LIN {X -32.888,Y -21.847,Z -39.181,A -90.000,B 90.000,C 0.000} C_DIS
LIN {X -32.646,Y -21.814,Z -39.101,A -90.000,B 90.000,C 0.000} C_DIS
LIN {X -32.451,Y -21.791,Z -39.046,A -90.000,B 90.000,C 0.000} C_DIS
LIN {X -32.080,Y -21.753,Z -38.957,A -90.000,B 90.000,C 0.000} C_DIS
LIN {X -31.853,Y -21.730,Z -38.910,A -90.000,B 90.000,C 0.000} C_DIS
LIN {X -31.718,Y -21.717,Z -38.887,A -90.000,B 90.000,C 0.000} C_DIS
LIN {X -31.508,Y -21.700,Z -38.859,A -90.000,B 90.000,C 0.000} C_DIS
LIN {X -31.116,Y -21.673,Z -38.819,A -90.000,B 90.000,C 0.000} C_DIS
LIN {X -31.063,Y -21.669,Z -38.814,A -90.000,B 90.000,C 0.000} C_DIS
LIN {X -30.892,Y -21.659,Z -38.806,A -90.000,B 90.000,C 0.000} C_DIS
LIN {X -30.823,Y -21.657,Z -38.806,A -90.000,B 90.000,C 0.000} C_DIS
LIN {X -30.549,Y -21.645,Z -38.800,A -90.000,B 90.000,C 0.000} C_DIS
LIN {X -30.055,Y -21.635,Z -38.810,A -90.000,B 90.000,C 0.000} C_DIS
LIN {X -28.776,Y -21.601,Z -38.842,A -90.000,B 90.000,C 0.000} C_DIS
LIN {X -28.195,Y -21.575,Z -38.837,A -90.000,B 90.000,C 0.000} C_DIS
LIN {X -27.943,Y -21.565,Z -38.836,A -90.000,B 90.000,C 0.000} C_DIS
LIN {X -27.045,Y -21.542,Z -38.826,A -90.000,B 90.000,C 0.000} C_DIS
LIN {X -26.882,Y -21.540,Z -38.829,A -90.000,B 90.000,C 0.000} C_DIS
LIN {X -26.670,Y -21.539,Z -38.837,A -90.000,B 90.000,C 0.000} C_DIS
LIN {X -26.459,Y -21.525,Z -38.814,A -90.000,B 90.000,C 0.000} C_DIS
LIN {X -26.307,Y -21.516,Z -38.801,A -90.000,B 90.000,C 0.000} C_DIS
LIN {X -26.029,Y -21.496,Z -38.784,A -90.000,B 90.000,C 0.000} C_DIS
LIN {X -25.788,Y -21.478,Z -38.772,A -90.000,B 90.000,C 0.000} C_DIS
LIN {X -25.199,Y -21.452,Z -38.736,A -90.000,B 90.000,C 0.000} C_DIS
LIN {X -24.907,Y -21.440,Z -38.729,A -90.000,B 90.000,C 0.000} C_DIS
LIN {X -24.488,Y -21.430,Z -38.731,A -90.000,B 90.000,C 0.000} C_DIS
LIN {X -24.339,Y -21.421,Z -38.722,A -90.000,B 90.000,C 0.000} C_DIS
LIN {X -23.648,Y -21.391,Z -38.698,A -90.000,B 90.000,C 0.000} C_DIS
LIN {X -22.784,Y -21.370,Z -38.662,A -90.000,B 90.000,C 0.000} C_DIS
LIN {X -22.360,Y -21.341,Z -38.605,A -90.000,B 90.000,C 0.000} C_DIS
LIN {X -22.032,Y -21.308,Z -38.567,A -90.000,B 90.000,C 0.000} C_DIS
LIN {X -22.032,Y -60.000,Z -38.567,A -90.000,B 90.000,C 0.000} C_DIS
LIN {X -41.599,Y -60.000,Z -38.134,A -90.000,B 90.000,C 0.000} C_DIS
LIN {X -41.599,Y -21.308,Z -38.134,A -90.000,B 90.000,C 0.000} C_DIS
LIN {X -40.454,Y -21.445,Z -38.400,A -90.000,B 90.000,C 0.000} C_DIS
LIN {X -39.852,Y -21.524,Z -38.553,A -90.000,B 90.000,C 0.000} C_DIS
LIN {X -39.336,Y -21.580,Z -38.649,A -90.000,B 90.000,C 0.000} C_DIS
LIN {X -38.632,Y -21.653,Z -38.787,A -90.000,B 90.000,C 0.000} C_DIS
LIN {X -37.790,Y -21.739,Z -38.950,A -90.000,B 90.000,C 0.000} C_DIS
LIN {X -36.979,Y -21.831,Z -39.143,A -90.000,B 90.000,C 0.000} C_DIS
LIN {X -36.858,Y -21.843,Z -39.172,A -90.000,B 90.000,C 0.000} C_DIS
LIN {X -36.574,Y -21.789,Z -38.973,A -90.000,B 90.000,C 0.000} C_DIS
LIN {X -36.491,Y -21.774,Z -38.918,A -90.000,B 90.000,C 0.000} C_DIS
LIN {X -36.292,Y -21.725,Z -38.792,A -90.000,B 90.000,C 0.000} C_DIS
LIN {X -36.111,Y -21.683,Z -38.685,A -90.000,B 90.000,C 0.000} C_DIS
LIN {X -34.878,Y -21.399,Z -38.007,A -90.000,B 90.000,C 0.000} C_DIS
LIN {X -34.510,Y -21.319,Z -37.820,A -90.000,B 90.000,C 0.000} C_DIS
LIN {X -34.454,Y -21.308,Z -37.795,A -90.000,B 90.000,C 0.000} C_DIS
LIN {X -34.454,Y -60.000,Z -37.795,A -90.000,B 90.000,C 0.000} C_DIS
LIN {X -100.614,Y -60.000,Z -38.290,A -90.000,B 90.000,C 0.000} C_DIS
LIN {X -100.614,Y -21.308,Z -38.290,A -90.000,B 90.000,C 0.000} C_DIS
LIN {X -100.205,Y -21.414,Z -38.194,A -90.000,B 90.000,C 0.000} C_DIS
LIN {X -100.106,Y -21.441,Z -38.173,A -90.000,B 90.000,C 0.000} C_DIS
LIN {X -100.009,Y -21.463,Z -38.155,A -90.000,B 90.000,C 0.000} C_DIS
LIN {X -99.788,Y -21.508,Z -38.090,A -90.000,B 90.000,C 0.000} C_DIS
LIN {X -99.614,Y -21.546,Z -38.045,A -90.000,B 90.000,C 0.000} C_DIS
LIN {X -99.380,Y -21.597,Z -37.989,A -90.000,B 90.000,C 0.000} C_DIS
LIN {X -99.127,Y -21.649,Z -37.935,A -90.000,B 90.000,C 0.000} C_DIS
LIN {X -98.699,Y -21.744,Z -37.869,A -90.000,B 90.000,C 0.000} C_DIS
LIN {X -98.267,Y -21.842,Z -37.814,A -90.000,B 90.000,C 0.000} C_DIS
LIN {X -98.126,Y -21.876,Z -37.800,A -90.000,B 90.000,C 0.000} C_DIS
LIN {X -98.086,Y -21.872,Z -37.753,A -90.000,B 90.000,C 0.000} C_DIS
LIN {X -98.019,Y -21.862,Z -37.682,A -90.000,B 90.000,C 0.000} C_DIS
LIN {X -97.690,Y -21.825,Z -37.351,A -90.000,B 90.000,C 0.000} C_DIS
LIN {X -97.548,Y -21.812,Z -37.215,A -90.000,B 90.000,C 0.000} C_DIS
LIN {X -97.502,Y -21.804,Z -37.162,A -90.000,B 90.000,C 0.000} C_DIS
LIN {X -97.462,Y -21.795,Z -37.117,A -90.000,B 90.000,C 0.000} C_DIS
LIN {X -97.361,Y -21.778,Z -37.014,A -90.000,B 90.000,C 0.000} C_DIS
LIN {X -97.077,Y -21.736,Z -36.733,A -90.000,B 90.000,C 0.000} C_DIS
LIN {X -96.910,Y -21.718,Z -36.582,A -90.000,B 90.000,C 0.000} C_DIS
LIN {X -96.744,Y -21.701,Z -36.444,A -90.000,B 90.000,C 0.000} C_DIS
LIN {X -96.611,Y -21.685,Z -36.336,A -90.000,B 90.000,C 0.000} C_DIS
LIN {X -96.274,Y -21.633,Z -36.025,A -90.000,B 90.000,C 0.000} C_DIS
LIN {X -96.149,Y -21.616,Z -35.917,A -90.000,B 90.000,C 0.000} C_DIS
LIN {X -96.043,Y -21.602,Z -35.833,A -90.000,B 90.000,C 0.000} C_DIS
LIN {X -95.731,Y -21.565,Z -35.597,A -90.000,B 90.000,C 0.000} C_DIS
LIN {X -95.458,Y -21.538,Z -35.389,A -90.000,B 90.000,C 0.000} C_DIS
LIN {X -95.333,Y -21.527,Z -35.300,A -90.000,B 90.000,C 0.000} C_DIS
LIN {X -95.028,Y -21.504,Z -35.104,A -90.000,B 90.000,C 0.000} C_DIS
LIN {X -94.893,Y -21.487,Z -35.002,A -90.000,B 90.000,C 0.000} C_DIS
LIN {X -94.794,Y -21.476,Z -34.928,A -90.000,B 90.000,C 0.000} C_DIS
LIN {X -94.672,Y -21.461,Z -34.843,A -90.000,B 90.000,C 0.000} C_DIS
LIN {X -94.553,Y -21.452,Z -34.767,A -90.000,B 90.000,C 0.000} C_DIS
LIN {X -94.476,Y -21.447,Z -34.719,A -90.000,B 90.000,C 0.000} C_DIS
LIN {X -94.315,Y -21.438,Z -34.624,A -90.000,B 90.000,C 0.000} C_DIS
LIN {X -94.176,Y -21.543,Z -34.477,A -90.000,B 90.000,C 0.000} C_DIS
LIN {X -94.101,Y -21.597,Z -34.407,A -90.000,B 90.000,C 0.000} C_DIS
LIN {X -94.045,Y -21.640,Z -34.344,A -90.000,B 90.000,C 0.000} C_DIS
LIN {X -93.974,Y -21.686,Z -34.273,A -90.000,B 90.000,C 0.000} C_DIS
LIN {X -93.825,Y -21.782,Z -34.136,A -90.000,B 90.000,C 0.000} C_DIS
LIN {X -93.634,Y -21.882,Z -33.989,A -90.000,B 90.000,C 0.000} C_DIS
LIN {X -93.528,Y -21.938,Z -33.912,A -90.000,B 90.000,C 0.000} C_DIS
LIN {X -93.397,Y -21.998,Z -33.825,A -90.000,B 90.000,C 0.000} C_DIS
LIN {X -93.347,Y -22.020,Z -33.794,A -90.000,B 90.000,C 0.000} C_DIS
LIN {X -93.262,Y -22.063,Z -33.743,A -90.000,B 90.000,C 0.000} C_DIS
LIN {X -93.192,Y -22.098,Z -33.703,A -90.000,B 90.000,C 0.000} C_DIS
LIN {X -93.048,Y -22.171,Z -33.612,A -90.000,B 90.000,C 0.000} C_DIS
LIN {X -92.988,Y -22.202,Z -33.559,A -90.000,B 90.000,C 0.000} C_DIS
LIN {X -92.889,Y -22.249,Z -33.478,A -90.000,B 90.000,C 0.000} C_DIS
LIN {X -92.767,Y -22.303,Z -33.387,A -90.000,B 90.000,C 0.000} C_DIS
LIN {X -92.764,Y -22.310,Z -33.201,A -90.000,B 90.000,C 0.000} C_DIS
LIN {X -92.753,Y -22.312,Z -33.050,A -90.000,B 90.000,C 0.000} C_DIS
LIN {X -92.734,Y -22.314,Z -32.891,A -90.000,B 90.000,C 0.000} C_DIS
LIN {X -92.716,Y -22.316,Z -32.752,A -90.000,B 90.000,C 0.000} C_DIS
LIN {X -92.695,Y -22.319,Z -32.637,A -90.000,B 90.000,C 0.000} C_DIS
LIN {X -92.629,Y -22.333,Z -32.322,A -90.000,B 90.000,C 0.000} C_DIS
LIN {X -92.598,Y -22.336,Z -32.198,A -90.000,B 90.000,C 0.000} C_DIS
LIN {X -92.561,Y -22.339,Z -32.070,A -90.000,B 90.000,C 0.000} C_DIS
LIN {X -92.530,Y -22.340,Z -31.975,A -90.000,B 90.000,C 0.000} C_DIS
LIN {X -92.451,Y -22.340,Z -31.766,A -90.000,B 90.000,C 0.000} C_DIS
LIN {X -92.397,Y -22.342,Z -31.640,A -90.000,B 90.000,C 0.000} C_DIS
LIN {X -92.293,Y -22.347,Z -31.422,A -90.000,B 90.000,C 0.000} C_DIS
LIN {X -92.165,Y -22.356,Z -31.181,A -90.000,B 90.000,C 0.000} C_DIS
LIN {X -92.072,Y -22.354,Z -31.025,A -90.000,B 90.000,C 0.000} C_DIS
LIN {X -92.020,Y -22.354,Z -30.944,A -90.000,B 90.000,C 0.000} C_DIS
LIN {X -91.933,Y -22.351,Z -30.824,A -90.000,B 90.000,C 0.000} C_DIS
LIN {X -91.750,Y -22.350,Z -30.588,A -90.000,B 90.000,C 0.000} C_DIS
LIN {X -91.667,Y -22.356,Z -30.485,A -90.000,B 90.000,C 0.000} C_DIS
LIN {X -91.552,Y -22.367,Z -30.354,A -90.000,B 90.000,C 0.000} C_DIS
LIN {X -91.426,Y -22.379,Z -30.212,A -90.000,B 90.000,C 0.000} C_DIS
LIN {X -91.373,Y -22.380,Z -30.154,A -90.000,B 90.000,C 0.000} C_DIS
LIN {X -91.227,Y -22.374,Z -29.968,A -90.000,B 90.000,C 0.000} C_DIS
LIN {X -91.132,Y -22.363,Z -29.854,A -90.000,B 90.000,C 0.000} C_DIS
LIN {X -91.028,Y -22.353,Z -29.740,A -90.000,B 90.000,C 0.000} C_DIS
LIN {X -90.920,Y -22.337,Z -29.632,A -90.000,B 90.000,C 0.000} C_DIS
LIN {X -90.736,Y -22.311,Z -29.456,A -90.000,B 90.000,C 0.000} C_DIS
LIN {X -90.615,Y -22.290,Z -29.351,A -90.000,B 90.000,C 0.000} C_DIS
LIN {X -90.528,Y -22.277,Z -29.280,A -90.000,B 90.000,C 0.000} C_DIS
LIN {X -90.420,Y -22.270,Z -29.195,A -90.000,B 90.000,C 0.000} C_DIS
LIN {X -90.287,Y -22.263,Z -29.095,A -90.000,B 90.000,C 0.000} C_DIS
LIN {X -90.131,Y -22.249,Z -28.995,A -90.000,B 90.000,C 0.000} C_DIS
LIN {X -90.003,Y -22.240,Z -28.917,A -90.000,B 90.000,C 0.000} C_DIS
LIN {X -89.988,Y -22.176,Z -28.780,A -90.000,B 90.000,C 0.000} C_DIS
LIN {X -89.968,Y -22.121,Z -28.658,A -90.000,B 90.000,C 0.000} C_DIS
LIN {X -89.961,Y -22.105,Z -28.627,A -90.000,B 90.000,C 0.000} C_DIS
LIN {X -89.926,Y -22.035,Z -28.465,A -90.000,B 90.000,C 0.000} C_DIS
LIN {X -89.879,Y -21.950,Z -28.270,A -90.000,B 90.000,C 0.000} C_DIS
LIN {X -89.848,Y -21.896,Z -28.172,A -90.000,B 90.000,C 0.000} C_DIS
LIN {X -89.820,Y -21.853,Z -28.089,A -90.000,B 90.000,C 0.000} C_DIS
LIN {X -89.771,Y -21.787,Z -27.950,A -90.000,B 90.000,C 0.000} C_DIS
LIN {X -89.722,Y -21.730,Z -27.825,A -90.000,B 90.000,C 0.000} C_DIS
LIN {X -89.648,Y -21.664,Z -27.633,A -90.000,B 90.000,C 0.000} C_DIS
LIN {X -89.586,Y -21.616,Z -27.488,A -90.000,B 90.000,C 0.000} C_DIS
LIN {X -89.533,Y -21.577,Z -27.378,A -90.000,B 90.000,C 0.000} C_DIS
LIN {X -89.338,Y -21.426,Z -27.003,A -90.000,B 90.000,C 0.000} C_DIS
LIN {X -89.314,Y -21.412,Z -26.959,A -90.000,B 90.000,C 0.000} C_DIS
LIN {X -89.215,Y -21.354,Z -26.785,A -90.000,B 90.000,C 0.000} C_DIS
LIN {X -89.141,Y -21.308,Z -26.675,A -90.000,B 90.000,C 0.000} C_DIS
LIN {X -89.043,Y -21.258,Z -26.529,A -90.000,B 90.000,C 0.000} C_DIS
LIN {X -88.953,Y -21.197,Z -26.391,A -90.000,B 90.000,C 0.000} C_DIS
LIN {X -88.870,Y -21.132,Z -26.262,A -90.000,B 90.000,C 0.000} C_DIS
LIN {X -88.725,Y -21.011,Z -26.027,A -90.000,B 90.000,C 0.000} C_DIS
LIN {X -88.663,Y -20.954,Z -25.922,A -90.000,B 90.000,C 0.000} C_DIS
LIN {X -88.608,Y -20.898,Z -25.824,A -90.000,B 90.000,C 0.000} C_DIS
LIN {X -88.559,Y -20.843,Z -25.734,A -90.000,B 90.000,C 0.000} C_DIS
LIN {X -88.517,Y -20.789,Z -25.652,A -90.000,B 90.000,C 0.000} C_DIS
LIN {X -88.482,Y -20.735,Z -25.576,A -90.000,B 90.000,C 0.000} C_DIS
LIN {X -88.452,Y -20.682,Z -25.509,A -90.000,B 90.000,C 0.000} C_DIS
LIN {X -88.429,Y -20.631,Z -25.448,A -90.000,B 90.000,C 0.000} C_DIS
LIN {X -88.405,Y -20.555,Z -25.369,A -90.000,B 90.000,C 0.000} C_DIS
LIN {X -88.394,Y -20.481,Z -25.306,A -90.000,B 90.000,C 0.000} C_DIS
LIN {X -88.394,Y -20.432,Z -25.273,A -90.000,B 90.000,C 0.000} C_DIS
LIN {X -88.405,Y -20.361,Z -25.234,A -90.000,B 90.000,C 0.000} C_DIS
LIN {X -88.411,Y -20.338,Z -25.225,A -90.000,B 90.000,C 0.000} C_DIS
LIN {X -88.427,Y -20.293,Z -25.210,A -90.000,B 90.000,C 0.000} C_DIS
LIN {X -88.461,Y -20.226,Z -25.199,A -90.000,B 90.000,C 0.000} C_DIS
LIN {X -88.490,Y -20.182,Z -25.200,A -90.000,B 90.000,C 0.000} C_DIS
LIN {X -88.542,Y -20.119,Z -25.211,A -90.000,B 90.000,C 0.000} C_DIS
LIN {X -88.583,Y -20.078,Z -25.225,A -90.000,B 90.000,C 0.000} C_DIS
LIN {X -88.628,Y -20.037,Z -25.245,A -90.000,B 90.000,C 0.000} C_DIS
LIN {X -88.678,Y -20.006,Z -25.270,A -90.000,B 90.000,C 0.000} C_DIS
LIN {X -88.732,Y -20.009,Z -25.301,A -90.000,B 90.000,C 0.000} C_DIS
LIN {X -88.853,Y -20.031,Z -25.377,A -90.000,B 90.000,C 0.000} C_DIS
LIN {X -88.919,Y -20.049,Z -25.422,A -90.000,B 90.000,C 0.000} C_DIS
LIN {X -89.063,Y -20.093,Z -25.526,A -90.000,B 90.000,C 0.000} C_DIS
LIN {X -89.222,Y -20.146,Z -25.648,A -90.000,B 90.000,C 0.000} C_DIS
LIN {X -89.306,Y -20.178,Z -25.715,A -90.000,B 90.000,C 0.000} C_DIS
LIN {X -89.577,Y -20.289,Z -25.941,A -90.000,B 90.000,C 0.000} C_DIS
LIN {X -89.773,Y -20.364,Z -26.110,A -90.000,B 90.000,C 0.000} C_DIS
LIN {X -89.979,Y -20.452,Z -26.292,A -90.000,B 90.000,C 0.000} C_DIS
LIN {X -90.194,Y -20.540,Z -26.487,A -90.000,B 90.000,C 0.000} C_DIS
LIN {X -90.418,Y -20.616,Z -26.694,A -90.000,B 90.000,C 0.000} C_DIS
LIN {X -90.649,Y -20.710,Z -26.911,A -90.000,B 90.000,C 0.000} C_DIS
LIN {X -90.887,Y -20.817,Z -27.138,A -90.000,B 90.000,C 0.000} C_DIS
LIN {X -91.130,Y -20.936,Z -27.373,A -90.000,B 90.000,C 0.000} C_DIS
LIN {X -91.378,Y -21.051,Z -27.616,A -90.000,B 90.000,C 0.000} C_DIS
LIN {X -91.630,Y -21.155,Z -27.865,A -90.000,B 90.000,C 0.000} C_DIS
LIN {X -91.884,Y -21.238,Z -28.119,A -90.000,B 90.000,C 0.000} C_DIS
LIN {X -92.140,Y -21.317,Z -28.378,A -90.000,B 90.000,C 0.000} C_DIS
LIN {X -92.396,Y -21.378,Z -28.640,A -90.000,B 90.000,C 0.000} C_DIS
LIN {X -92.653,Y -21.409,Z -28.905,A -90.000,B 90.000,C 0.000} C_DIS
LIN {X -92.908,Y -21.422,Z -29.171,A -90.000,B 90.000,C 0.000} C_DIS
LIN {X -93.160,Y -21.434,Z -29.437,A -90.000,B 90.000,C 0.000} C_DIS
LIN {X -93.410,Y -21.433,Z -29.703,A -90.000,B 90.000,C 0.000} C_DIS
LIN {X -93.655,Y -21.410,Z -29.966,A -90.000,B 90.000,C 0.000} C_DIS
LIN {X -93.895,Y -21.378,Z -30.227,A -90.000,B 90.000,C 0.000} C_DIS
LIN {X -94.129,Y -21.339,Z -30.485,A -90.000,B 90.000,C 0.000} C_DIS
LIN {X -94.356,Y -21.286,Z -30.737,A -90.000,B 90.000,C 0.000} C_DIS
LIN {X -94.575,Y -21.223,Z -30.984,A -90.000,B 90.000,C 0.000} C_DIS
LIN {X -94.785,Y -21.178,Z -31.223,A -90.000,B 90.000,C 0.000} C_DIS
LIN {X -94.984,Y -21.118,Z -31.455,A -90.000,B 90.000,C 0.000} C_DIS
LIN {X -95.173,Y -21.054,Z -31.678,A -90.000,B 90.000,C 0.000} C_DIS
LIN {X -95.350,Y -21.002,Z -31.891,A -90.000,B 90.000,C 0.000} C_DIS
LIN {X -95.514,Y -20.945,Z -32.093,A -90.000,B 90.000,C 0.000} C_DIS
LIN {X -95.664,Y -20.878,Z -32.284,A -90.000,B 90.000,C 0.000} C_DIS
LIN {X -95.733,Y -20.843,Z -32.374,A -90.000,B 90.000,C 0.000} C_DIS
LIN {X -95.860,Y -20.778,Z -32.544,A -90.000,B 90.000,C 0.000} C_DIS
LIN {X -95.971,Y -20.725,Z -32.700,A -90.000,B 90.000,C 0.000} C_DIS
LIN {X -96.064,Y -20.677,Z -32.840,A -90.000,B 90.000,C 0.000} C_DIS
LIN {X -96.139,Y -20.634,Z -32.964,A -90.000,B 90.000,C 0.000} C_DIS
LIN {X -96.195,Y -20.598,Z -33.070,A -90.000,B 90.000,C 0.000} C_DIS
LIN {X -96.215,Y -20.583,Z -33.116,A -90.000,B 90.000,C 0.000} C_DIS
LIN {X -96.240,Y -20.564,Z -33.194,A -90.000,B 90.000,C 0.000} C_DIS
LIN {X -96.245,Y -20.558,Z -33.239,A -90.000,B 90.000,C 0.000} C_DIS
LIN {X -96.241,Y -20.558,Z -33.263,A -90.000,B 90.000,C 0.000} C_DIS
LIN {X -96.237,Y -20.560,Z -33.273,A -90.000,B 90.000,C 0.000} C_DIS
LIN {X -96.224,Y -20.567,Z -33.288,A -90.000,B 90.000,C 0.000} C_DIS
LIN {X -96.216,Y -20.572,Z -33.294,A -90.000,B 90.000,C 0.000} C_DIS
LIN {X -96.181,Y -20.594,Z -33.303,A -90.000,B 90.000,C 0.000} C_DIS
LIN {X -96.150,Y -20.614,Z -33.301,A -90.000,B 90.000,C 0.000} C_DIS
LIN {X -96.113,Y -20.638,Z -33.294,A -90.000,B 90.000,C 0.000} C_DIS
LIN {X -96.070,Y -20.666,Z -33.280,A -90.000,B 90.000,C 0.000} C_DIS
LIN {X -95.963,Y -20.736,Z -33.235,A -90.000,B 90.000,C 0.000} C_DIS
LIN {X -95.830,Y -20.820,Z -33.163,A -90.000,B 90.000,C 0.000} C_DIS
LIN {X -95.668,Y -20.912,Z -33.065,A -90.000,B 90.000,C 0.000} C_DIS
LIN {X -95.477,Y -21.008,Z -32.939,A -90.000,B 90.000,C 0.000} C_DIS
LIN {X -95.257,Y -21.115,Z -32.784,A -90.000,B 90.000,C 0.000} C_DIS
LIN {X -95.005,Y -21.249,Z -32.600,A -90.000,B 90.000,C 0.000} C_DIS
LIN {X -94.867,Y -21.308,Z -32.496,A -90.000,B 90.000,C 0.000} C_DIS
LIN {X -94.735,Y -21.374,Z -32.395,A -90.000,B 90.000,C 0.000} C_DIS
LIN {X -94.474,Y -21.482,Z -32.210,A -90.000,B 90.000,C 0.000} C_DIS
LIN {X -94.461,Y -21.488,Z -32.201,A -90.000,B 90.000,C 0.000} C_DIS
LIN {X -94.382,Y -21.488,Z -31.861,A -90.000,B 90.000,C 0.000} C_DIS
LIN {X -94.318,Y -21.493,Z -31.618,A -90.000,B 90.000,C 0.000} C_DIS
LIN {X -94.247,Y -21.487,Z -31.407,A -90.000,B 90.000,C 0.000} C_DIS
LIN {X -94.177,Y -21.484,Z -31.221,A -90.000,B 90.000,C 0.000} C_DIS
LIN {X -94.106,Y -21.482,Z -31.041,A -90.000,B 90.000,C 0.000} C_DIS
LIN {X -94.015,Y -21.484,Z -30.835,A -90.000,B 90.000,C 0.000} C_DIS
LIN {X -93.966,Y -21.486,Z -30.734,A -90.000,B 90.000,C 0.000} C_DIS
LIN {X -93.872,Y -21.482,Z -30.551,A -90.000,B 90.000,C 0.000} C_DIS
LIN {X -93.807,Y -21.480,Z -30.436,A -90.000,B 90.000,C 0.000} C_DIS
LIN {X -93.713,Y -21.472,Z -30.276,A -90.000,B 90.000,C 0.000} C_DIS
LIN {X -93.592,Y -21.465,Z -30.076,A -90.000,B 90.000,C 0.000} C_DIS
LIN {X -93.524,Y -21.465,Z -29.969,A -90.000,B 90.000,C 0.000} C_DIS
LIN {X -93.480,Y -21.467,Z -29.903,A -90.000,B 90.000,C 0.000} C_DIS
LIN {X -93.350,Y -21.464,Z -29.726,A -90.000,B 90.000,C 0.000} C_DIS
LIN {X -93.271,Y -21.464,Z -29.624,A -90.000,B 90.000,C 0.000} C_DIS
LIN {X -93.117,Y -21.449,Z -29.439,A -90.000,B 90.000,C 0.000} C_DIS
LIN {X -93.016,Y -21.442,Z -29.324,A -90.000,B 90.000,C 0.000} C_DIS
LIN {X -92.865,Y -21.435,Z -29.167,A -90.000,B 90.000,C 0.000} C_DIS
LIN {X -92.717,Y -21.430,Z -29.015,A -90.000,B 90.000,C 0.000} C_DIS
LIN {X -92.650,Y -21.420,Z -28.936,A -90.000,B 90.000,C 0.000} C_DIS
LIN {X -92.474,Y -21.391,Z -28.734,A -90.000,B 90.000,C 0.000} C_DIS
LIN {X -92.283,Y -21.358,Z -28.541,A -90.000,B 90.000,C 0.000} C_DIS
LIN {X -92.197,Y -21.344,Z -28.455,A -90.000,B 90.000,C 0.000} C_DIS
LIN {X -92.033,Y -21.308,Z -28.310,A -90.000,B 90.000,C 0.000} C_DIS
LIN {X -92.033,Y -60.000,Z -28.310,A -90.000,B 90.000,C 0.000} C_DIS
LIN {X -106.753,Y -60.000,Z -42.835,A -90.000,B 90.000,C 0.000} C_DIS
LIN {X -106.753,Y -21.308,Z -42.835,A -90.000,B 90.000,C 0.000} C_DIS
LIN {X -106.698,Y -21.320,Z -42.690,A -90.000,B 90.000,C 0.000} C_DIS
LIN {X -106.625,Y -21.329,Z -42.511,A -90.000,B 90.000,C 0.000} C_DIS
LIN {X -106.563,Y -21.338,Z -42.376,A -90.000,B 90.000,C 0.000} C_DIS
LIN {X -106.515,Y -21.344,Z -42.278,A -90.000,B 90.000,C 0.000} C_DIS
LIN {X -106.418,Y -21.361,Z -42.101,A -90.000,B 90.000,C 0.000} C_DIS
LIN {X -106.303,Y -21.371,Z -41.904,A -90.000,B 90.000,C 0.000} C_DIS
LIN {X -106.128,Y -21.381,Z -41.620,A -90.000,B 90.000,C 0.000} C_DIS
LIN {X -106.072,Y -21.384,Z -41.530,A -90.000,B 90.000,C 0.000} C_DIS
LIN {X -105.932,Y -21.384,Z -41.327,A -90.000,B 90.000,C 0.000} C_DIS
LIN {X -105.884,Y -21.388,Z -41.261,A -90.000,B 90.000,C 0.000} C_DIS
LIN {X -105.762,Y -21.391,Z -41.111,A -90.000,B 90.000,C 0.000} C_DIS
LIN {X -105.660,Y -21.396,Z -40.990,A -90.000,B 90.000,C 0.000} C_DIS
LIN {X -105.461,Y -21.388,Z -40.772,A -90.000,B 90.000,C 0.000} C_DIS
LIN {X -105.340,Y -21.384,Z -40.641,A -90.000,B 90.000,C 0.000} C_DIS
LIN {X -105.188,Y -21.379,Z -40.480,A -90.000,B 90.000,C 0.000} C_DIS
LIN {X -105.077,Y -21.369,Z -40.379,A -90.000,B 90.000,C 0.000} C_DIS
LIN {X -104.931,Y -21.359,Z -40.252,A -90.000,B 90.000,C 0.000} C_DIS
LIN {X -104.638,Y -21.339,Z -40.023,A -90.000,B 90.000,C 0.000} C_DIS
LIN {X -104.496,Y -21.324,Z -39.921,A -90.000,B 90.000,C 0.000} C_DIS
LIN {X -104.322,Y -21.308,Z -39.805,A -90.000,B 90.000,C 0.000} C_DIS
LIN {X -104.322,Y -60.000,Z -39.805,A -90.000,B 90.000,C 0.000} C_DIS
LIN {X -105.044,Y -60.000,Z -54.822,A -90.000,B 90.000,C 0.000} C_DIS
LIN {X -105.044,Y -21.308,Z -54.822,A -90.000,B 90.000,C 0.000} C_DIS
LIN {X -105.069,Y -21.321,Z -54.621,A -90.000,B 90.000,C 0.000} C_DIS
LIN {X -105.095,Y -21.338,Z -54.365,A -90.000,B 90.000,C 0.000} C_DIS
LIN {X -105.108,Y -21.349,Z -54.203,A -90.000,B 90.000,C 0.000} C_DIS
LIN {X -105.120,Y -21.370,Z -53.971,A -90.000,B 90.000,C 0.000} C_DIS
LIN {X -105.123,Y -21.397,Z -53.738,A -90.000,B 90.000,C 0.000} C_DIS
LIN {X -105.123,Y -21.401,Z -53.704,A -90.000,B 90.000,C 0.000} C_DIS
LIN {X -105.093,Y -21.442,Z -53.157,A -90.000,B 90.000,C 0.000} C_DIS
LIN {X -105.069,Y -21.467,Z -52.818,A -90.000,B 90.000,C 0.000} C_DIS
LIN {X -105.063,Y -21.473,Z -52.761,A -90.000,B 90.000,C 0.000} C_DIS
LIN {X -105.048,Y -21.477,Z -52.667,A -90.000,B 90.000,C 0.000} C_DIS
LIN {X -105.149,Y -21.407,Z -52.427,A -90.000,B 90.000,C 0.000} C_DIS
LIN {X -105.259,Y -21.331,Z -52.151,A -90.000,B 90.000,C 0.000} C_DIS
LIN {X -105.294,Y -21.308,Z -52.064,A -90.000,B 90.000,C 0.000} C_DIS
LIN {X -105.294,Y -60.000,Z -52.064,A -90.000,B 90.000,C 0.000} C_DIS
LIN {X -106.298,Y -60.000,Z -243.561,A -90.000,B 90.000,C 0.000} C_DIS
LIN {X -106.298,Y -21.308,Z -243.561,A -90.000,B 90.000,C 0.000} C_DIS
LIN {X -103.088,Y -21.308,Z -241.440,A -90.000,B 90.000,C 0.000} C_DIS
LIN {X -99.816,Y -21.308,Z -239.308,A -90.000,B 90.000,C 0.000} C_DIS
LIN {X -95.252,Y -21.308,Z -236.320,A -90.000,B 90.000,C 0.000} C_DIS
LIN {X -91.143,Y -21.308,Z -233.668,A -90.000,B 90.000,C 0.000} C_DIS
LIN {X -87.088,Y -21.308,Z -231.059,A -90.000,B 90.000,C 0.000} C_DIS
LIN {X -82.371,Y -21.308,Z -228.080,A -90.000,B 90.000,C 0.000} C_DIS
LIN {X -81.805,Y -21.308,Z -227.726,A -90.000,B 90.000,C 0.000} C_DIS
LIN {X -78.607,Y -21.308,Z -225.688,A -90.000,B 90.000,C 0.000} C_DIS
LIN {X -73.743,Y -21.308,Z -222.667,A -90.000,B 90.000,C 0.000} C_DIS
LIN {X -72.906,Y -21.308,Z -222.152,A -90.000,B 90.000,C 0.000} C_DIS
LIN {X -70.393,Y -21.308,Z -220.553,A -90.000,B 90.000,C 0.000} C_DIS
LIN {X -65.618,Y -21.308,Z -217.528,A -90.000,B 90.000,C 0.000} C_DIS
LIN {X -62.348,Y -21.308,Z -215.481,A -90.000,B 90.000,C 0.000} C_DIS
LIN {X -57.206,Y -21.308,Z -212.204,A -90.000,B 90.000,C 0.000} C_DIS
LIN {X -54.876,Y -21.308,Z -210.688,A -90.000,B 90.000,C 0.000} C_DIS
LIN {X -53.612,Y -21.308,Z -209.828,A -90.000,B 90.000,C 0.000} C_DIS
LIN {X -51.750,Y -21.308,Z -208.571,A -90.000,B 90.000,C 0.000} C_DIS
LIN {X -48.408,Y -21.308,Z -206.325,A -90.000,B 90.000,C 0.000} C_DIS
LIN {X -43.930,Y -21.308,Z -203.053,A -90.000,B 90.000,C 0.000} C_DIS
LIN {X -43.271,Y -21.308,Z -202.576,A -90.000,B 90.000,C 0.000} C_DIS
LIN {X -41.226,Y -21.308,Z -200.972,A -90.000,B 90.000,C 0.000} C_DIS
LIN {X -38.879,Y -21.308,Z -199.146,A -90.000,B 90.000,C 0.000} C_DIS
LIN {X -36.934,Y -21.308,Z -197.549,A -90.000,B 90.000,C 0.000} C_DIS
LIN {X -35.130,Y -21.308,Z -196.075,A -90.000,B 90.000,C 0.000} C_DIS
LIN {X -34.778,Y -21.308,Z -195.785,A -90.000,B 90.000,C 0.000} C_DIS
LIN {X -31.882,Y -21.308,Z -193.355,A -90.000,B 90.000,C 0.000} C_DIS
LIN {X -29.706,Y -21.308,Z -191.547,A -90.000,B 90.000,C 0.000} C_DIS
LIN {X -28.831,Y -21.308,Z -190.838,A -90.000,B 90.000,C 0.000} C_DIS
LIN {X -26.880,Y -21.308,Z -189.191,A -90.000,B 90.000,C 0.000} C_DIS
LIN {X -25.951,Y -21.308,Z -188.426,A -90.000,B 90.000,C 0.000} C_DIS
LIN {X -24.127,Y -21.308,Z -186.810,A -90.000,B 90.000,C 0.000} C_DIS
LIN {X -23.356,Y -21.308,Z -186.146,A -90.000,B 90.000,C 0.000} C_DIS
LIN {X -21.765,Y -21.308,Z -184.625,A -90.000,B 90.000,C 0.000} C_DIS
LIN {X -20.866,Y -21.308,Z -183.794,A -90.000,B 90.000,C 0.000} C_DIS
LIN {X -19.977,Y -21.308,Z -182.891,A -90.000,B 90.000,C 0.000} C_DIS
LIN {X -18.317,Y -21.308,Z -181.146,A -90.000,B 90.000,C 0.000} C_DIS
LIN {X -17.573,Y -21.308,Z -180.310,A -90.000,B 90.000,C 0.000} C_DIS
LIN {X -16.056,Y -21.308,Z -178.540,A -90.000,B 90.000,C 0.000} C_DIS
LIN {X -15.581,Y -21.308,Z -177.947,A -90.000,B 90.000,C 0.000} C_DIS
LIN {X -13.815,Y -21.308,Z -175.626,A -90.000,B 90.000,C 0.000} C_DIS
LIN {X -13.433,Y -21.308,Z -175.084,A -90.000,B 90.000,C 0.000} C_DIS
LIN {X -12.010,Y -21.308,Z -172.920,A -90.000,B 90.000,C 0.000} C_DIS
LIN {X -11.581,Y -21.308,Z -172.209,A -90.000,B 90.000,C 0.000} C_DIS
LIN {X -10.371,Y -21.308,Z -169.988,A -90.000,B 90.000,C 0.000} C_DIS
LIN {X -10.195,Y -21.308,Z -169.626,A -90.000,B 90.000,C 0.000} C_DIS
LIN {X -9.156,Y -21.308,Z -167.174,A -90.000,B 90.000,C 0.000} C_DIS
LIN {X -8.450,Y -21.308,Z -164.687,A -90.000,B 90.000,C 0.000} C_DIS
LIN {X -8.260,Y -21.308,Z -162.882,A -90.000,B 90.000,C 0.000} C_DIS
LIN {X -8.458,Y -21.308,Z -161.763,A -90.000,B 90.000,C 0.000} C_DIS
LIN {X -8.472,Y -21.308,Z -161.636,A -90.000,B 90.000,C 0.000} C_DIS
LIN {X -8.769,Y -21.308,Z -161.034,A -90.000,B 90.000,C 0.000} C_DIS
LIN {X -8.856,Y -21.308,Z -160.833,A -90.000,B 90.000,C 0.000} C_DIS
LIN {X -9.036,Y -21.308,Z -160.615,A -90.000,B 90.000,C 0.000} C_DIS
LIN {X -9.306,Y -21.308,Z -160.266,A -90.000,B 90.000,C 0.000} C_DIS
LIN {X -9.545,Y -21.308,Z -159.939,A -90.000,B 90.000,C 0.000} C_DIS
LIN {X -9.686,Y -21.308,Z -159.808,A -90.000,B 90.000,C 0.000} C_DIS
LIN {X -9.852,Y -21.308,Z -159.644,A -90.000,B 90.000,C 0.000} C_DIS
LIN {X -10.574,Y -21.308,Z -158.896,A -90.000,B 90.000,C 0.000} C_DIS
LIN {X -11.850,Y -21.308,Z -157.687,A -90.000,B 90.000,C 0.000} C_DIS
LIN {X -11.980,Y -21.308,Z -157.573,A -90.000,B 90.000,C 0.000} C_DIS
LIN {X -12.609,Y -21.308,Z -157.005,A -90.000,B 90.000,C 0.000} C_DIS
LIN {X -13.539,Y -21.308,Z -156.145,A -90.000,B 90.000,C 0.000} C_DIS
LIN {X -15.141,Y -21.308,Z -154.736,A -90.000,B 90.000,C 0.000} C_DIS
LIN {X -15.479,Y -21.308,Z -154.434,A -90.000,B 90.000,C 0.000} C_DIS
LIN {X -17.805,Y -21.308,Z -152.418,A -90.000,B 90.000,C 0.000} C_DIS
LIN {X -18.003,Y -21.308,Z -152.245,A -90.000,B 90.000,C 0.000} C_DIS
LIN {X -20.742,Y -21.308,Z -149.905,A -90.000,B 90.000,C 0.000} C_DIS
LIN {X -23.986,Y -21.308,Z -146.969,A -90.000,B 90.000,C 0.000} C_DIS
LIN {X -24.449,Y -21.308,Z -146.500,A -90.000,B 90.000,C 0.000} C_DIS
LIN {X -27.291,Y -21.308,Z -143.601,A -90.000,B 90.000,C 0.000} C_DIS
LIN {X -27.577,Y -21.308,Z -143.304,A -90.000,B 90.000,C 0.000} C_DIS
LIN {X -29.792,Y -21.308,Z -140.601,A -90.000,B 90.000,C 0.000} C_DIS
LIN {X -30.581,Y -21.308,Z -139.636,A -90.000,B 90.000,C 0.000} C_DIS
LIN {X -30.866,Y -21.308,Z -139.266,A -90.000,B 90.000,C 0.000} C_DIS
LIN {X -33.340,Y -21.308,Z -135.307,A -90.000,B 90.000,C 0.000} C_DIS
LIN {X -33.584,Y -21.308,Z -134.908,A -90.000,B 90.000,C 0.000} C_DIS
LIN {X -34.739,Y -21.308,Z -132.640,A -90.000,B 90.000,C 0.000} C_DIS
LIN {X -35.802,Y -21.308,Z -130.571,A -90.000,B 90.000,C 0.000} C_DIS
LIN {X -36.367,Y -21.308,Z -129.339,A -90.000,B 90.000,C 0.000} C_DIS
LIN {X -38.010,Y -21.308,Z -126.340,A -90.000,B 90.000,C 0.000} C_DIS
LIN {X -38.234,Y -21.308,Z -125.927,A -90.000,B 90.000,C 0.000} C_DIS
LIN {X -38.830,Y -21.308,Z -124.589,A -90.000,B 90.000,C 0.000} C_DIS
LIN {X -39.775,Y -21.308,Z -122.705,A -90.000,B 90.000,C 0.000} C_DIS
LIN {X -40.134,Y -21.308,Z -121.942,A -90.000,B 90.000,C 0.000} C_DIS
LIN {X -40.428,Y -21.308,Z -121.319,A -90.000,B 90.000,C 0.000} C_DIS
LIN {X -40.536,Y -21.308,Z -121.131,A -90.000,B 90.000,C 0.000} C_DIS
LIN {X -41.229,Y -21.308,Z -119.875,A -90.000,B 90.000,C 0.000} C_DIS
LIN {X -41.479,Y -21.308,Z -119.499,A -90.000,B 90.000,C 0.000} C_DIS
LIN {X -42.251,Y -21.308,Z -118.243,A -90.000,B 90.000,C 0.000} C_DIS
LIN {X -42.755,Y -21.308,Z -117.565,A -90.000,B 90.000,C 0.000} C_DIS
LIN {X -43.528,Y -21.308,Z -116.448,A -90.000,B 90.000,C 0.000} C_DIS
LIN {X -43.729,Y -21.308,Z -116.189,A -90.000,B 90.000,C 0.000} C_DIS
LIN {X -44.373,Y -21.308,Z -115.345,A -90.000,B 90.000,C 0.000} C_DIS
LIN {X -45.324,Y -21.308,Z -114.074,A -90.000,B 90.000,C 0.000} C_DIS
LIN {X -45.866,Y -21.308,Z -113.383,A -90.000,B 90.000,C 0.000} C_DIS
LIN {X -47.168,Y -21.308,Z -111.690,A -90.000,B 90.000,C 0.000} C_DIS
LIN {X -47.630,Y -21.308,Z -111.081,A -90.000,B 90.000,C 0.000} C_DIS
LIN {X -49.173,Y -21.308,Z -109.053,A -90.000,B 90.000,C 0.000} C_DIS
LIN {X -50.151,Y -21.308,Z -107.783,A -90.000,B 90.000,C 0.000} C_DIS
LIN {X -50.848,Y -21.308,Z -106.858,A -90.000,B 90.000,C 0.000} C_DIS
LIN {X -52.123,Y -21.308,Z -105.206,A -90.000,B 90.000,C 0.000} C_DIS
LIN {X -52.607,Y -21.308,Z -104.565,A -90.000,B 90.000,C 0.000} C_DIS
LIN {X -52.745,Y -21.308,Z -104.387,A -90.000,B 90.000,C 0.000} C_DIS
LIN {X -54.154,Y -21.308,Z -102.475,A -90.000,B 90.000,C 0.000} C_DIS
LIN {X -55.267,Y -21.308,Z -101.017,A -90.000,B 90.000,C 0.000} C_DIS
LIN {X -55.765,Y -21.308,Z -100.339,A -90.000,B 90.000,C 0.000} C_DIS
LIN {X -56.691,Y -21.308,Z -99.122,A -90.000,B 90.000,C 0.000} C_DIS
LIN {X -57.351,Y -21.308,Z -98.226,A -90.000,B 90.000,C 0.000} C_DIS
LIN {X -57.685,Y -21.308,Z -97.788,A -90.000,B 90.000,C 0.000} C_DIS
LIN {X -58.913,Y -21.308,Z -96.140,A -90.000,B 90.000,C 0.000} C_DIS
LIN {X -59.964,Y -21.308,Z -94.774,A -90.000,B 90.000,C 0.000} C_DIS
LIN {X -60.459,Y -21.308,Z -94.126,A -90.000,B 90.000,C 0.000} C_DIS
LIN {X -61.689,Y -21.308,Z -92.563,A -90.000,B 90.000,C 0.000} C_DIS
LIN {X -61.979,Y -21.308,Z -92.183,A -90.000,B 90.000,C 0.000} C_DIS
LIN {X -62.075,Y -21.308,Z -92.061,A -90.000,B 90.000,C 0.000} C_DIS
LIN {X -62.273,Y -21.308,Z -91.820,A -90.000,B 90.000,C 0.000} C_DIS
LIN {X -63.792,Y -21.308,Z -89.940,A -90.000,B 90.000,C 0.000} C_DIS
LIN {X -64.607,Y -21.308,Z -89.000,A -90.000,B 90.000,C 0.000} C_DIS
LIN {X -65.508,Y -21.308,Z -87.940,A -90.000,B 90.000,C 0.000} C_DIS
LIN {X -66.973,Y -21.308,Z -86.326,A -90.000,B 90.000,C 0.000} C_DIS
LIN {X -67.261,Y -21.308,Z -86.004,A -90.000,B 90.000,C 0.000} C_DIS
LIN {X -68.067,Y -21.308,Z -85.147,A -90.000,B 90.000,C 0.000} C_DIS
LIN {X -69.004,Y -21.308,Z -84.137,A -90.000,B 90.000,C 0.000} C_DIS
LIN {X -69.387,Y -21.308,Z -83.735,A -90.000,B 90.000,C 0.000} C_DIS
LIN {X -70.788,Y -21.308,Z -82.252,A -90.000,B 90.000,C 0.000} C_DIS
LIN {X -71.941,Y -21.308,Z -81.076,A -90.000,B 90.000,C 0.000} C_DIS
LIN {X -72.392,Y -21.308,Z -80.620,A -90.000,B 90.000,C 0.000} C_DIS
LIN {X -73.095,Y -21.308,Z -79.946,A -90.000,B 90.000,C 0.000} C_DIS
LIN {X -73.838,Y -21.308,Z -79.252,A -90.000,B 90.000,C 0.000} C_DIS
LIN {X -74.456,Y -21.308,Z -78.730,A -90.000,B 90.000,C 0.000} C_DIS
LIN {X -74.785,Y -21.308,Z -78.470,A -90.000,B 90.000,C 0.000} C_DIS
LIN {X -74.879,Y -21.308,Z -78.412,A -90.000,B 90.000,C 0.000} C_DIS
LIN {X -75.195,Y -21.308,Z -78.252,A -90.000,B 90.000,C 0.000} C_DIS
LIN {X -75.630,Y -21.308,Z -78.126,A -90.000,B 90.000,C 0.000} C_DIS
LIN {X -75.787,Y -21.308,Z -78.087,A -90.000,B 90.000,C 0.000} C_DIS
LIN {X -76.056,Y -21.308,Z -78.047,A -90.000,B 90.000,C 0.000} C_DIS
LIN {X -76.894,Y -21.308,Z -77.930,A -90.000,B 90.000,C 0.000} C_DIS
LIN {X -77.355,Y -21.308,Z -77.854,A -90.000,B 90.000,C 0.000} C_DIS
LIN {X -77.849,Y -21.308,Z -77.730,A -90.000,B 90.000,C 0.000} C_DIS
LIN {X -78.579,Y -21.308,Z -77.541,A -90.000,B 90.000,C 0.000} C_DIS
LIN {X -79.013,Y -21.308,Z -77.412,A -90.000,B 90.000,C 0.000} C_DIS
LIN {X -79.736,Y -21.308,Z -77.130,A -90.000,B 90.000,C 0.000} C_DIS
LIN {X -80.170,Y -21.308,Z -76.958,A -90.000,B 90.000,C 0.000} C_DIS
LIN {X -80.547,Y -21.308,Z -76.788,A -90.000,B 90.000,C 0.000} C_DIS
LIN {X -80.897,Y -21.308,Z -76.614,A -90.000,B 90.000,C 0.000} C_DIS
LIN {X -81.332,Y -21.308,Z -76.382,A -90.000,B 90.000,C 0.000} C_DIS
LIN {X -82.505,Y -21.308,Z -75.693,A -90.000,B 90.000,C 0.000} C_DIS
LIN {X -82.676,Y -21.308,Z -75.583,A -90.000,B 90.000,C 0.000} C_DIS
LIN {X -83.081,Y -21.308,Z -75.309,A -90.000,B 90.000,C 0.000} C_DIS
LIN {X -84.324,Y -21.308,Z -74.384,A -90.000,B 90.000,C 0.000} C_DIS
LIN {X -84.704,Y -21.308,Z -74.064,A -90.000,B 90.000,C 0.000} C_DIS
LIN {X -85.524,Y -21.308,Z -73.360,A -90.000,B 90.000,C 0.000} C_DIS
LIN {X -85.989,Y -21.308,Z -73.008,A -90.000,B 90.000,C 0.000} C_DIS
LIN {X -86.331,Y -21.308,Z -72.718,A -90.000,B 90.000,C 0.000} C_DIS
LIN {X -86.709,Y -21.308,Z -72.405,A -90.000,B 90.000,C 0.000} C_DIS
LIN {X -87.534,Y -21.308,Z -71.748,A -90.000,B 90.000,C 0.000} C_DIS
LIN {X -88.217,Y -21.308,Z -71.189,A -90.000,B 90.000,C 0.000} C_DIS
LIN {X -88.473,Y -21.308,Z -70.971,A -90.000,B 90.000,C 0.000} C_DIS
LIN {X -89.025,Y -21.308,Z -70.445,A -90.000,B 90.000,C 0.000} C_DIS
LIN {X -89.698,Y -21.308,Z -69.759,A -90.000,B 90.000,C 0.000} C_DIS
LIN {X -90.218,Y -21.308,Z -69.233,A -90.000,B 90.000,C 0.000} C_DIS
LIN {X -90.915,Y -21.308,Z -68.576,A -90.000,B 90.000,C 0.000} C_DIS
LIN {X -91.488,Y -21.308,Z -68.094,A -90.000,B 90.000,C 0.000} C_DIS
LIN {X -92.255,Y -21.308,Z -67.488,A -90.000,B 90.000,C 0.000} C_DIS
LIN {X -93.159,Y -21.308,Z -66.783,A -90.000,B 90.000,C 0.000} C_DIS
LIN {X -94.056,Y -21.308,Z -66.064,A -90.000,B 90.000,C 0.000} C_DIS
LIN {X -94.167,Y -21.308,Z -65.973,A -90.000,B 90.000,C 0.000} C_DIS
LIN {X -95.356,Y -21.308,Z -64.955,A -90.000,B 90.000,C 0.000} C_DIS
LIN {X -96.022,Y -21.308,Z -64.371,A -90.000,B 90.000,C 0.000} C_DIS
LIN {X -96.838,Y -21.308,Z -63.673,A -90.000,B 90.000,C 0.000} C_DIS
LIN {X -97.560,Y -21.308,Z -63.093,A -90.000,B 90.000,C 0.000} C_DIS
LIN {X -98.592,Y -21.308,Z -62.345,A -90.000,B 90.000,C 0.000} C_DIS
LIN {X -99.274,Y -21.308,Z -61.871,A -90.000,B 90.000,C 0.000} C_DIS
LIN {X -99.631,Y -21.308,Z -61.610,A -90.000,B 90.000,C 0.000} C_DIS
LIN {X -100.266,Y -21.308,Z -61.131,A -90.000,B 90.000,C 0.000} C_DIS
LIN {X -100.609,Y -21.308,Z -60.872,A -90.000,B 90.000,C 0.000} C_DIS
LIN {X -101.087,Y -21.308,Z -60.479,A -90.000,B 90.000,C 0.000} C_DIS
LIN {X -101.747,Y -21.308,Z -59.928,A -90.000,B 90.000,C 0.000} C_DIS
LIN {X -101.991,Y -21.308,Z -59.697,A -90.000,B 90.000,C 0.000} C_DIS
LIN {X -102.204,Y -21.308,Z -59.488,A -90.000,B 90.000,C 0.000} C_DIS
LIN {X -102.880,Y -21.308,Z -58.737,A -90.000,B 90.000,C 0.000} C_DIS
LIN {X -102.927,Y -21.308,Z -58.681,A -90.000,B 90.000,C 0.000} C_DIS
LIN {X -103.289,Y -21.308,Z -58.204,A -90.000,B 90.000,C 0.000} C_DIS
LIN {X -103.597,Y -21.308,Z -57.807,A -90.000,B 90.000,C 0.000} C_DIS
LIN {X -103.810,Y -21.308,Z -57.522,A -90.000,B 90.000,C 0.000} C_DIS
LIN {X -103.897,Y -21.308,Z -57.394,A -90.000,B 90.000,C 0.000} C_DIS
LIN {X -104.096,Y -21.308,Z -57.044,A -90.000,B 90.000,C 0.000} C_DIS
LIN {X -104.326,Y -21.308,Z -56.628,A -90.000,B 90.000,C 0.000} C_DIS
LIN {X -104.506,Y -21.308,Z -56.283,A -90.000,B 90.000,C 0.000} C_DIS
LIN {X -104.526,Y -21.308,Z -56.241,A -90.000,B 90.000,C 0.000} C_DIS
LIN {X -104.692,Y -21.308,Z -55.830,A -90.000,B 90.000,C 0.000} C_DIS
LIN {X -104.819,Y -21.308,Z -55.524,A -90.000,B 90.000,C 0.000} C_DIS
LIN {X -104.950,Y -21.308,Z -55.168,A -90.000,B 90.000,C 0.000} C_DIS
LIN {X -105.022,Y -21.308,Z -54.920,A -90.000,B 90.000,C 0.000} C_DIS
LIN {X -105.066,Y -21.308,Z -54.726,A -90.000,B 90.000,C 0.000} C_DIS
LIN {X -105.127,Y -21.308,Z -54.423,A -90.000,B 90.000,C 0.000} C_DIS
LIN {X -105.169,Y -21.308,Z -54.195,A -90.000,B 90.000,C 0.000} C_DIS
LIN {X -105.198,Y -21.308,Z -54.055,A -90.000,B 90.000,C 0.000} C_DIS
LIN {X -105.283,Y -21.308,Z -53.589,A -90.000,B 90.000,C 0.000} C_DIS
LIN {X -105.308,Y -21.308,Z -53.178,A -90.000,B 90.000,C 0.000} C_DIS
LIN {X -105.317,Y -21.308,Z -52.845,A -90.000,B 90.000,C 0.000} C_DIS
LIN {X -105.332,Y -21.308,Z -52.573,A -90.000,B 90.000,C 0.000} C_DIS
LIN {X -105.301,Y -21.308,Z -52.182,A -90.000,B 90.000,C 0.000} C_DIS
LIN {X -105.287,Y -21.308,Z -51.966,A -90.000,B 90.000,C 0.000} C_DIS
LIN {X -105.258,Y -21.308,Z -51.634,A -90.000,B 90.000,C 0.000} C_DIS
LIN {X -105.254,Y -21.308,Z -51.608,A -90.000,B 90.000,C 0.000} C_DIS
LIN {X -105.175,Y -21.308,Z -51.271,A -90.000,B 90.000,C 0.000} C_DIS
LIN {X -105.014,Y -21.308,Z -50.654,A -90.000,B 90.000,C 0.000} C_DIS
LIN {X -104.889,Y -21.308,Z -50.360,A -90.000,B 90.000,C 0.000} C_DIS
LIN {X -104.719,Y -21.308,Z -50.089,A -90.000,B 90.000,C 0.000} C_DIS
LIN {X -104.657,Y -21.308,Z -50.008,A -90.000,B 90.000,C 0.000} C_DIS
LIN {X -104.687,Y -21.308,Z -49.968,A -90.000,B 90.000,C 0.000} C_DIS
LIN {X -105.061,Y -21.308,Z -49.430,A -90.000,B 90.000,C 0.000} C_DIS
LIN {X -105.624,Y -21.308,Z -48.564,A -90.000,B 90.000,C 0.000} C_DIS
LIN {X -105.643,Y -21.308,Z -48.532,A -90.000,B 90.000,C 0.000} C_DIS
LIN {X -105.876,Y -21.308,Z -48.081,A -90.000,B 90.000,C 0.000} C_DIS
LIN {X -106.064,Y -21.308,Z -47.701,A -90.000,B 90.000,C 0.000} C_DIS
LIN {X -106.251,Y -21.308,Z -47.251,A -90.000,B 90.000,C 0.000} C_DIS
LIN {X -106.530,Y -21.308,Z -46.532,A -90.000,B 90.000,C 0.000} C_DIS
LIN {X -106.676,Y -21.308,Z -46.028,A -90.000,B 90.000,C 0.000} C_DIS
LIN {X -106.759,Y -21.308,Z -45.731,A -90.000,B 90.000,C 0.000} C_DIS
LIN {X -106.853,Y -21.308,Z -45.283,A -90.000,B 90.000,C 0.000} C_DIS
LIN {X -106.878,Y -21.308,Z -45.106,A -90.000,B 90.000,C 0.000} C_DIS
LIN {X -106.909,Y -21.308,Z -44.861,A -90.000,B 90.000,C 0.000} C_DIS
LIN {X -106.927,Y -21.308,Z -44.655,A -90.000,B 90.000,C 0.000} C_DIS
LIN {X -106.943,Y -21.308,Z -44.416,A -90.000,B 90.000,C 0.000} C_DIS
LIN {X -106.942,Y -21.308,Z -44.369,A -90.000,B 90.000,C 0.000} C_DIS
LIN {X -106.934,Y -21.308,Z -44.069,A -90.000,B 90.000,C 0.000} C_DIS
LIN {X -106.917,Y -21.308,Z -43.690,A -90.000,B 90.000,C 0.000} C_DIS
LIN {X -106.793,Y -21.308,Z -42.992,A -90.000,B 90.000,C 0.000} C_DIS
LIN {X -106.713,Y -21.308,Z -42.678,A -90.000,B 90.000,C 0.000} C_DIS
LIN {X -106.671,Y -21.308,Z -42.549,A -90.000,B 90.000,C 0.000} C_DIS
LIN {X -106.612,Y -21.308,Z -42.377,A -90.000,B 90.000,C 0.000} C_DIS
LIN {X -106.485,Y -21.308,Z -42.049,A -90.000,B 90.000,C 0.000} C_DIS
LIN {X -106.430,Y -21.308,Z -41.933,A -90.000,B 90.000,C 0.000} C_DIS
LIN {X -106.342,Y -21.308,Z -41.763,A -90.000,B 90.000,C 0.000} C_DIS
LIN {X -106.171,Y -21.308,Z -41.456,A -90.000,B 90.000,C 0.000} C_DIS
LIN {X -106.045,Y -21.308,Z -41.274,A -90.000,B 90.000,C 0.000} C_DIS
LIN {X -105.988,Y -21.308,Z -41.184,A -90.000,B 90.000,C 0.000} C_DIS
LIN {X -105.775,Y -21.308,Z -40.904,A -90.000,B 90.000,C 0.000} C_DIS
LIN {X -105.587,Y -21.308,Z -40.716,A -90.000,B 90.000,C 0.000} C_DIS
LIN {X -105.534,Y -21.308,Z -40.657,A -90.000,B 90.000,C 0.000} C_DIS
LIN {X -105.283,Y -21.308,Z -40.411,A -90.000,B 90.000,C 0.000} C_DIS
LIN {X -105.000,Y -21.308,Z -40.203,A -90.000,B 90.000,C 0.000} C_DIS
LIN {X -104.705,Y -21.308,Z -40.012,A -90.000,B 90.000,C 0.000} C_DIS
LIN {X -104.680,Y -21.308,Z -39.994,A -90.000,B 90.000,C 0.000} C_DIS
LIN {X -104.370,Y -21.308,Z -39.828,A -90.000,B 90.000,C 0.000} C_DIS
LIN {X -104.303,Y -21.308,Z -39.797,A -90.000,B 90.000,C 0.000} C_DIS
LIN {X -103.966,Y -21.308,Z -39.675,A -90.000,B 90.000,C 0.000} C_DIS
LIN {X -103.728,Y -21.308,Z -39.594,A -90.000,B 90.000,C 0.000} C_DIS
LIN {X -103.597,Y -21.308,Z -39.555,A -90.000,B 90.000,C 0.000} C_DIS
LIN {X -103.259,Y -21.308,Z -39.446,A -90.000,B 90.000,C 0.000} C_DIS
LIN {X -102.889,Y -21.308,Z -39.368,A -90.000,B 90.000,C 0.000} C_DIS
LIN {X -102.620,Y -21.308,Z -39.330,A -90.000,B 90.000,C 0.000} C_DIS
LIN {X -102.129,Y -21.308,Z -39.279,A -90.000,B 90.000,C 0.000} C_DIS
LIN {X -101.542,Y -21.308,Z -39.226,A -90.000,B 90.000,C 0.000} C_DIS
LIN {X -101.335,Y -21.308,Z -39.218,A -90.000,B 90.000,C 0.000} C_DIS
LIN {X -101.225,Y -21.308,Z -39.067,A -90.000,B 90.000,C 0.000} C_DIS
LIN {X -101.011,Y -21.308,Z -38.780,A -90.000,B 90.000,C 0.000} C_DIS
LIN {X -100.825,Y -21.308,Z -38.540,A -90.000,B 90.000,C 0.000} C_DIS
LIN {X -100.594,Y -21.308,Z -38.266,A -90.000,B 90.000,C 0.000} C_DIS
LIN {X -100.384,Y -21.308,Z -38.025,A -90.000,B 90.000,C 0.000} C_DIS
LIN {X -100.073,Y -21.308,Z -37.742,A -90.000,B 90.000,C 0.000} C_DIS
LIN {X -99.605,Y -21.308,Z -37.353,A -90.000,B 90.000,C 0.000} C_DIS
LIN {X -99.111,Y -21.308,Z -36.995,A -90.000,B 90.000,C 0.000} C_DIS
LIN {X -99.001,Y -21.308,Z -36.923,A -90.000,B 90.000,C 0.000} C_DIS
LIN {X -98.624,Y -21.308,Z -36.688,A -90.000,B 90.000,C 0.000} C_DIS
LIN {X -98.358,Y -21.308,Z -36.526,A -90.000,B 90.000,C 0.000} C_DIS
LIN {X -98.244,Y -21.308,Z -36.454,A -90.000,B 90.000,C 0.000} C_DIS
LIN {X -98.005,Y -21.308,Z -36.311,A -90.000,B 90.000,C 0.000} C_DIS
LIN {X -97.434,Y -21.308,Z -35.989,A -90.000,B 90.000,C 0.000} C_DIS
LIN {X -97.132,Y -21.308,Z -35.829,A -90.000,B 90.000,C 0.000} C_DIS
LIN {X -96.747,Y -21.308,Z -35.600,A -90.000,B 90.000,C 0.000} C_DIS
LIN {X -96.229,Y -21.308,Z -35.323,A -90.000,B 90.000,C 0.000} C_DIS
LIN {X -96.053,Y -21.308,Z -35.233,A -90.000,B 90.000,C 0.000} C_DIS
LIN {X -95.808,Y -21.308,Z -35.102,A -90.000,B 90.000,C 0.000} C_DIS
LIN {X -95.398,Y -21.308,Z -34.903,A -90.000,B 90.000,C 0.000} C_DIS
LIN {X -95.159,Y -21.308,Z -34.781,A -90.000,B 90.000,C 0.000} C_DIS
LIN {X -94.897,Y -21.308,Z -34.657,A -90.000,B 90.000,C 0.000} C_DIS
LIN {X -94.617,Y -21.308,Z -34.520,A -90.000,B 90.000,C 0.000} C_DIS
LIN {X -94.674,Y -21.308,Z -34.375,A -90.000,B 90.000,C 0.000} C_DIS
LIN {X -94.789,Y -21.308,Z -34.052,A -90.000,B 90.000,C 0.000} C_DIS
LIN {X -94.859,Y -21.308,Z -33.708,A -90.000,B 90.000,C 0.000} C_DIS
LIN {X -94.876,Y -21.308,Z -33.537,A -90.000,B 90.000,C 0.000} C_DIS
LIN {X -94.897,Y -21.308,Z -33.218,A -90.000,B 90.000,C 0.000} C_DIS
LIN {X -94.892,Y -21.308,Z -33.135,A -90.000,B 90.000,C 0.000} C_DIS
LIN {X -94.882,Y -21.308,Z -32.991,A -90.000,B 90.000,C 0.000} C_DIS
LIN {X -94.887,Y -21.308,Z -32.783,A -90.000,B 90.000,C 0.000} C_DIS
LIN {X -94.884,Y -21.308,Z -32.677,A -90.000,B 90.000,C 0.000} C_DIS
LIN {X -94.855,Y -21.308,Z -32.359,A -90.000,B 90.000,C 0.000} C_DIS
LIN {X -94.772,Y -21.308,Z -32.037,A -90.000,B 90.000,C 0.000} C_DIS
LIN {X -94.724,Y -21.308,Z -31.892,A -90.000,B 90.000,C 0.000} C_DIS
LIN {X -94.642,Y -21.308,Z -31.536,A -90.000,B 90.000,C 0.000} C_DIS
LIN {X -94.515,Y -21.308,Z -31.208,A -90.000,B 90.000,C 0.000} C_DIS
LIN {X -94.451,Y -21.308,Z -31.085,A -90.000,B 90.000,C 0.000} C_DIS
LIN {X -94.278,Y -21.308,Z -30.657,A -90.000,B 90.000,C 0.000} C_DIS
LIN {X -94.106,Y -21.308,Z -30.351,A -90.000,B 90.000,C 0.000} C_DIS
LIN {X -94.060,Y -21.308,Z -30.286,A -90.000,B 90.000,C 0.000} C_DIS
LIN {X -93.832,Y -21.308,Z -29.915,A -90.000,B 90.000,C 0.000} C_DIS
LIN {X -93.791,Y -21.308,Z -29.855,A -90.000,B 90.000,C 0.000} C_DIS
LIN {X -93.577,Y -21.308,Z -29.577,A -90.000,B 90.000,C 0.000} C_DIS
LIN {X -93.316,Y -21.308,Z -29.321,A -90.000,B 90.000,C 0.000} C_DIS
LIN {X -92.920,Y -21.308,Z -28.947,A -90.000,B 90.000,C 0.000} C_DIS
LIN {X -92.549,Y -21.308,Z -28.639,A -90.000,B 90.000,C 0.000} C_DIS
LIN {X -92.237,Y -21.308,Z -28.423,A -90.000,B 90.000,C 0.000} C_DIS
LIN {X -92.204,Y -21.308,Z -28.402,A -90.000,B 90.000,C 0.000} C_DIS
LIN {X -91.627,Y -21.308,Z -28.090,A -90.000,B 90.000,C 0.000} C_DIS
LIN {X -91.290,Y -21.308,Z -27.917,A -90.000,B 90.000,C 0.000} C_DIS
LIN {X -91.002,Y -21.308,Z -27.783,A -90.000,B 90.000,C 0.000} C_DIS
LIN {X -90.673,Y -21.308,Z -27.663,A -90.000,B 90.000,C 0.000} C_DIS
LIN {X -90.605,Y -21.308,Z -27.628,A -90.000,B 90.000,C 0.000} C_DIS
LIN {X -90.230,Y -21.308,Z -27.461,A -90.000,B 90.000,C 0.000} C_DIS
LIN {X -89.870,Y -21.308,Z -27.233,A -90.000,B 90.000,C 0.000} C_DIS
LIN {X -89.372,Y -21.308,Z -26.852,A -90.000,B 90.000,C 0.000} C_DIS
LIN {X -89.342,Y -21.308,Z -26.826,A -90.000,B 90.000,C 0.000} C_DIS
LIN {X -88.801,Y -21.308,Z -26.420,A -90.000,B 90.000,C 0.000} C_DIS
LIN {X -88.566,Y -21.308,Z -26.231,A -90.000,B 90.000,C 0.000} C_DIS
LIN {X -88.126,Y -21.308,Z -25.915,A -90.000,B 90.000,C 0.000} C_DIS
LIN {X -87.570,Y -21.308,Z -25.490,A -90.000,B 90.000,C 0.000} C_DIS
LIN {X -87.485,Y -21.308,Z -25.420,A -90.000,B 90.000,C 0.000} C_DIS
LIN {X -86.884,Y -21.308,Z -24.954,A -90.000,B 90.000,C 0.000} C_DIS
LIN {X -86.219,Y -21.308,Z -24.390,A -90.000,B 90.000,C 0.000} C_DIS
LIN {X -85.746,Y -21.308,Z -23.949,A -90.000,B 90.000,C 0.000} C_DIS
LIN {X -85.241,Y -21.308,Z -23.419,A -90.000,B 90.000,C 0.000} C_DIS
LIN {X -84.638,Y -21.308,Z -22.736,A -90.000,B 90.000,C 0.000} C_DIS
LIN {X -84.142,Y -21.308,Z -22.171,A -90.000,B 90.000,C 0.000} C_DIS
LIN {X -83.653,Y -21.308,Z -21.641,A -90.000,B 90.000,C 0.000} C_DIS
LIN {X -83.191,Y -21.308,Z -21.163,A -90.000,B 90.000,C 0.000} C_DIS
LIN {X -83.064,Y -21.308,Z -21.035,A -90.000,B 90.000,C 0.000} C_DIS
LIN {X -82.749,Y -21.308,Z -20.752,A -90.000,B 90.000,C 0.000} C_DIS
LIN {X -82.599,Y -21.308,Z -20.623,A -90.000,B 90.000,C 0.000} C_DIS
LIN {X -82.278,Y -21.308,Z -20.365,A -90.000,B 90.000,C 0.000} C_DIS
LIN {X -81.874,Y -21.308,Z -20.057,A -90.000,B 90.000,C 0.000} C_DIS
LIN {X -81.541,Y -21.308,Z -19.830,A -90.000,B 90.000,C 0.000} C_DIS
LIN {X -81.158,Y -21.308,Z -19.633,A -90.000,B 90.000,C 0.000} C_DIS
LIN {X -81.135,Y -21.308,Z -19.622,A -90.000,B 90.000,C 0.000} C_DIS
LIN {X -80.989,Y -21.308,Z -19.566,A -90.000,B 90.000,C 0.000} C_DIS
LIN {X -80.356,Y -21.308,Z -19.333,A -90.000,B 90.000,C 0.000} C_DIS
LIN {X -80.123,Y -21.308,Z -19.276,A -90.000,B 90.000,C 0.000} C_DIS
LIN {X -79.835,Y -21.308,Z -19.214,A -90.000,B 90.000,C 0.000} C_DIS
LIN {X -79.163,Y -21.308,Z -19.149,A -90.000,B 90.000,C 0.000} C_DIS
LIN {X -78.970,Y -21.308,Z -19.134,A -90.000,B 90.000,C 0.000} C_DIS
LIN {X -78.773,Y -21.308,Z -19.138,A -90.000,B 90.000,C 0.000} C_DIS
LIN {X -78.580,Y -21.308,Z -19.149,A -90.000,B 90.000,C 0.000} C_DIS
LIN {X -77.961,Y -21.308,Z -19.225,A -90.000,B 90.000,C 0.000} C_DIS
LIN {X -77.930,Y -21.308,Z -19.228,A -90.000,B 90.000,C 0.000} C_DIS
LIN {X -77.765,Y -21.308,Z -19.255,A -90.000,B 90.000,C 0.000} C_DIS
LIN {X -77.611,Y -21.308,Z -19.284,A -90.000,B 90.000,C 0.000} C_DIS
LIN {X -77.260,Y -21.308,Z -19.370,A -90.000,B 90.000,C 0.000} C_DIS
LIN {X -76.878,Y -21.308,Z -19.490,A -90.000,B 90.000,C 0.000} C_DIS
LIN {X -76.518,Y -21.308,Z -19.608,A -90.000,B 90.000,C 0.000} C_DIS
LIN {X -76.280,Y -21.308,Z -19.701,A -90.000,B 90.000,C 0.000} C_DIS
LIN {X -75.771,Y -21.308,Z -19.943,A -90.000,B 90.000,C 0.000} C_DIS
LIN {X -75.430,Y -21.308,Z -20.107,A -90.000,B 90.000,C 0.000} C_DIS
LIN {X -75.324,Y -21.308,Z -20.164,A -90.000,B 90.000,C 0.000} C_DIS
LIN {X -74.720,Y -21.308,Z -20.526,A -90.000,B 90.000,C 0.000} C_DIS
LIN {X -74.616,Y -21.308,Z -20.589,A -90.000,B 90.000,C 0.000} C_DIS
LIN {X -74.358,Y -21.308,Z -20.760,A -90.000,B 90.000,C 0.000} C_DIS
LIN {X -73.616,Y -21.308,Z -21.268,A -90.000,B 90.000,C 0.000} C_DIS
LIN {X -73.189,Y -21.308,Z -21.582,A -90.000,B 90.000,C 0.000} C_DIS
LIN {X -72.909,Y -21.308,Z -21.794,A -90.000,B 90.000,C 0.000} C_DIS
LIN {X -72.471,Y -21.308,Z -22.140,A -90.000,B 90.000,C 0.000} C_DIS
LIN {X -72.278,Y -21.308,Z -22.307,A -90.000,B 90.000,C 0.000} C_DIS
LIN {X -71.548,Y -21.308,Z -22.959,A -90.000,B 90.000,C 0.000} C_DIS
LIN {X -71.300,Y -21.308,Z -23.209,A -90.000,B 90.000,C 0.000} C_DIS
LIN {X -70.619,Y -21.308,Z -23.937,A -90.000,B 90.000,C 0.000} C_DIS
LIN {X -70.419,Y -21.308,Z -24.154,A -90.000,B 90.000,C 0.000} C_DIS
LIN {X -70.209,Y -21.308,Z -24.436,A -90.000,B 90.000,C 0.000} C_DIS
LIN {X -70.019,Y -21.308,Z -24.711,A -90.000,B 90.000,C 0.000} C_DIS
LIN {X -69.482,Y -21.308,Z -25.586,A -90.000,B 90.000,C 0.000} C_DIS
LIN {X -69.315,Y -21.308,Z -25.895,A -90.000,B 90.000,C 0.000} C_DIS
LIN {X -69.019,Y -21.308,Z -26.695,A -90.000,B 90.000,C 0.000} C_DIS
LIN {X -68.818,Y -21.308,Z -27.325,A -90.000,B 90.000,C 0.000} C_DIS
LIN {X -68.725,Y -21.308,Z -27.666,A -90.000,B 90.000,C 0.000} C_DIS
LIN {X -68.651,Y -21.308,Z -28.009,A -90.000,B 90.000,C 0.000} C_DIS
LIN {X -68.404,Y -21.308,Z -29.419,A -90.000,B 90.000,C 0.000} C_DIS
LIN {X -68.390,Y -21.308,Z -29.554,A -90.000,B 90.000,C 0.000} C_DIS
LIN {X -68.342,Y -21.308,Z -29.813,A -90.000,B 90.000,C 0.000} C_DIS
LIN {X -68.169,Y -21.308,Z -30.838,A -90.000,B 90.000,C 0.000} C_DIS
LIN {X -67.739,Y -21.308,Z -31.909,A -90.000,B 90.000,C 0.000} C_DIS
LIN {X -66.931,Y -21.308,Z -32.724,A -90.000,B 90.000,C 0.000} C_DIS
LIN {X -66.667,Y -21.308,Z -33.008,A -90.000,B 90.000,C 0.000} C_DIS
LIN {X -65.551,Y -21.308,Z -33.742,A -90.000,B 90.000,C 0.000} C_DIS
LIN {X -64.893,Y -21.308,Z -34.162,A -90.000,B 90.000,C 0.000} C_DIS
LIN {X -62.586,Y -21.308,Z -35.372,A -90.000,B 90.000,C 0.000} C_DIS
LIN {X -61.966,Y -21.308,Z -35.659,A -90.000,B 90.000,C 0.000} C_DIS
LIN {X -60.116,Y -21.308,Z -36.499,A -90.000,B 90.000,C 0.000} C_DIS
LIN {X -57.848,Y -21.308,Z -37.449,A -90.000,B 90.000,C 0.000} C_DIS
LIN {X -55.476,Y -21.308,Z -38.341,A -90.000,B 90.000,C 0.000} C_DIS
LIN {X -55.206,Y -21.308,Z -38.441,A -90.000,B 90.000,C 0.000} C_DIS
LIN {X -54.253,Y -21.308,Z -38.756,A -90.000,B 90.000,C 0.000} C_DIS
LIN {X -52.455,Y -21.308,Z -39.322,A -90.000,B 90.000,C 0.000} C_DIS
LIN {X -51.382,Y -21.308,Z -39.621,A -90.000,B 90.000,C 0.000} C_DIS
LIN {X -49.520,Y -21.308,Z -40.117,A -90.000,B 90.000,C 0.000} C_DIS
LIN {X -49.416,Y -21.308,Z -40.143,A -90.000,B 90.000,C 0.000} C_DIS
LIN {X -46.926,Y -21.308,Z -40.667,A -90.000,B 90.000,C 0.000} C_DIS
LIN {X -46.018,Y -21.308,Z -40.728,A -90.000,B 90.000,C 0.000} C_DIS
LIN {X -45.829,Y -21.308,Z -40.589,A -90.000,B 90.000,C 0.000} C_DIS
LIN {X -45.665,Y -21.308,Z -40.497,A -90.000,B 90.000,C 0.000} C_DIS
LIN {X -45.526,Y -21.308,Z -40.434,A -90.000,B 90.000,C 0.000} C_DIS
LIN {X -45.232,Y -21.308,Z -40.022,A -90.000,B 90.000,C 0.000} C_DIS
LIN {X -45.074,Y -21.308,Z -39.858,A -90.000,B 90.000,C 0.000} C_DIS
LIN {X -44.886,Y -21.308,Z -39.718,A -90.000,B 90.000,C 0.000} C_DIS
LIN {X -44.860,Y -21.308,Z -39.706,A -90.000,B 90.000,C 0.000} C_DIS
LIN {X -44.809,Y -21.308,Z -39.660,A -90.000,B 90.000,C 0.000} C_DIS
LIN {X -44.591,Y -21.308,Z -39.498,A -90.000,B 90.000,C 0.000} C_DIS
LIN {X -44.336,Y -21.308,Z -39.318,A -90.000,B 90.000,C 0.000} C_DIS
LIN {X -44.319,Y -21.308,Z -39.291,A -90.000,B 90.000,C 0.000} C_DIS
LIN {X -44.167,Y -21.308,Z -39.118,A -90.000,B 90.000,C 0.000} C_DIS
LIN {X -43.978,Y -21.308,Z -38.975,A -90.000,B 90.000,C 0.000} C_DIS
LIN {X -43.763,Y -21.308,Z -38.876,A -90.000,B 90.000,C 0.000} C_DIS
LIN {X -42.881,Y -21.308,Z -38.660,A -90.000,B 90.000,C 0.000} C_DIS
LIN {X -42.431,Y -21.308,Z -38.397,A -90.000,B 90.000,C 0.000} C_DIS
LIN {X -42.216,Y -21.308,Z -38.298,A -90.000,B 90.000,C 0.000} C_DIS
LIN {X -41.622,Y -21.308,Z -38.137,A -90.000,B 90.000,C 0.000} C_DIS
LIN {X -41.342,Y -21.308,Z -38.105,A -90.000,B 90.000,C 0.000} C_DIS
LIN {X -40.347,Y -21.308,Z -38.013,A -90.000,B 90.000,C 0.000} C_DIS
LIN {X -38.589,Y -21.308,Z -37.824,A -90.000,B 90.000,C 0.000} C_DIS
LIN {X -37.734,Y -21.308,Z -37.799,A -90.000,B 90.000,C 0.000} C_DIS
LIN {X -36.662,Y -21.308,Z -37.784,A -90.000,B 90.000,C 0.000} C_DIS
LIN {X -33.609,Y -21.308,Z -37.799,A -90.000,B 90.000,C 0.000} C_DIS
LIN {X -33.035,Y -21.308,Z -37.832,A -90.000,B 90.000,C 0.000} C_DIS
LIN {X -30.528,Y -21.308,Z -38.043,A -90.000,B 90.000,C 0.000} C_DIS
LIN {X -28.180,Y -21.308,Z -38.193,A -90.000,B 90.000,C 0.000} C_DIS
LIN {X -28.011,Y -21.308,Z -38.208,A -90.000,B 90.000,C 0.000} C_DIS
LIN {X -27.848,Y -21.308,Z -38.217,A -90.000,B 90.000,C 0.000} C_DIS
LIN {X -27.559,Y -21.308,Z -38.242,A -90.000,B 90.000,C 0.000} C_DIS
LIN {X -25.757,Y -21.308,Z -38.425,A -90.000,B 90.000,C 0.000} C_DIS
LIN {X -24.480,Y -21.308,Z -38.464,A -90.000,B 90.000,C 0.000} C_DIS
LIN {X -23.630,Y -21.308,Z -38.517,A -90.000,B 90.000,C 0.000} C_DIS
LIN {X -22.557,Y -21.308,Z -38.530,A -90.000,B 90.000,C 0.000} C_DIS
LIN {X -21.359,Y -21.308,Z -38.614,A -90.000,B 90.000,C 0.000} C_DIS
LIN {X -21.013,Y -21.308,Z -38.641,A -90.000,B 90.000,C 0.000} C_DIS
LIN {X -20.809,Y -21.308,Z -38.659,A -90.000,B 90.000,C 0.000} C_DIS
LIN {X -18.528,Y -21.308,Z -38.911,A -90.000,B 90.000,C 0.000} C_DIS
LIN {X -16.062,Y -21.308,Z -39.223,A -90.000,B 90.000,C 0.000} C_DIS
LIN {X -15.747,Y -21.308,Z -39.275,A -90.000,B 90.000,C 0.000} C_DIS
LIN {X -13.787,Y -21.308,Z -39.671,A -90.000,B 90.000,C 0.000} C_DIS
LIN {X -12.919,Y -21.308,Z -39.869,A -90.000,B 90.000,C 0.000} C_DIS
LIN {X -12.388,Y -21.308,Z -39.983,A -90.000,B 90.000,C 0.000} C_DIS
LIN {X -10.991,Y -21.308,Z -40.339,A -90.000,B 90.000,C 0.000} C_DIS
LIN {X -9.238,Y -21.308,Z -40.767,A -90.000,B 90.000,C 0.000} C_DIS
LIN {X -9.143,Y -21.308,Z -40.793,A -90.000,B 90.000,C 0.000} C_DIS
LIN {X -6.318,Y -21.308,Z -41.652,A -90.000,B 90.000,C 0.000} C_DIS
LIN {X -5.808,Y -21.308,Z -41.814,A -90.000,B 90.000,C 0.000} C_DIS
LIN {X -4.131,Y -21.308,Z -42.421,A -90.000,B 90.000,C 0.000} C_DIS
LIN {X -2.989,Y -21.308,Z -42.831,A -90.000,B 90.000,C 0.000} C_DIS
LIN {X -2.617,Y -21.308,Z -42.985,A -90.000,B 90.000,C 0.000} C_DIS
LIN {X -0.290,Y -21.308,Z -43.986,A -90.000,B 90.000,C 0.000} C_DIS
LIN {X 1.677,Y -21.308,Z -44.916,A -90.000,B 90.000,C 0.000} C_DIS
LIN {X 1.949,Y -21.308,Z -45.041,A -90.000,B 90.000,C 0.000} C_DIS
LIN {X 2.456,Y -21.308,Z -45.261,A -90.000,B 90.000,C 0.000} C_DIS
LIN {X 2.555,Y -21.308,Z -45.298,A -90.000,B 90.000,C 0.000} C_DIS
LIN {X 2.916,Y -21.308,Z -45.451,A -90.000,B 90.000,C 0.000} C_DIS
LIN {X 3.695,Y -21.308,Z -45.534,A -90.000,B 90.000,C 0.000} C_DIS
LIN {X 4.219,Y -21.308,Z -45.609,A -90.000,B 90.000,C 0.000} C_DIS
LIN {X 4.396,Y -21.308,Z -45.617,A -90.000,B 90.000,C 0.000} C_DIS
LIN {X 5.025,Y -21.308,Z -45.539,A -90.000,B 90.000,C 0.000} C_DIS
LIN {X 5.945,Y -21.308,Z -45.320,A -90.000,B 90.000,C 0.000} C_DIS
LIN {X 6.195,Y -21.308,Z -45.278,A -90.000,B 90.000,C 0.000} C_DIS
LIN {X 6.360,Y -21.308,Z -45.248,A -90.000,B 90.000,C 0.000} C_DIS
LIN {X 7.668,Y -21.308,Z -44.913,A -90.000,B 90.000,C 0.000} C_DIS
LIN {X 7.967,Y -21.308,Z -44.843,A -90.000,B 90.000,C 0.000} C_DIS
LIN {X 8.368,Y -21.308,Z -44.754,A -90.000,B 90.000,C 0.000} C_DIS
LIN {X 8.950,Y -21.308,Z -44.588,A -90.000,B 90.000,C 0.000} C_DIS
LIN {X 9.261,Y -21.308,Z -44.516,A -90.000,B 90.000,C 0.000} C_DIS
LIN {X 9.922,Y -21.308,Z -44.374,A -90.000,B 90.000,C 0.000} C_DIS
LIN {X 11.006,Y -21.308,Z -44.186,A -90.000,B 90.000,C 0.000} C_DIS
LIN {X 11.386,Y -21.308,Z -44.118,A -90.000,B 90.000,C 0.000} C_DIS
LIN {X 13.104,Y -21.308,Z -43.913,A -90.000,B 90.000,C 0.000} C_DIS
LIN {X 13.225,Y -21.308,Z -43.902,A -90.000,B 90.000,C 0.000} C_DIS
LIN {X 13.601,Y -21.308,Z -43.873,A -90.000,B 90.000,C 0.000} C_DIS
LIN {X 13.684,Y -21.308,Z -43.869,A -90.000,B 90.000,C 0.000} C_DIS
LIN {X 15.534,Y -21.308,Z -43.745,A -90.000,B 90.000,C 0.000} C_DIS
LIN {X 15.899,Y -21.308,Z -43.723,A -90.000,B 90.000,C 0.000} C_DIS
LIN {X 16.389,Y -21.308,Z -43.703,A -90.000,B 90.000,C 0.000} C_DIS
LIN {X 18.540,Y -21.308,Z -43.592,A -90.000,B 90.000,C 0.000} C_DIS
LIN {X 19.883,Y -21.308,Z -43.521,A -90.000,B 90.000,C 0.000} C_DIS
LIN {X 20.717,Y -21.308,Z -43.488,A -90.000,B 90.000,C 0.000} C_DIS
LIN {X 21.651,Y -21.308,Z -43.411,A -90.000,B 90.000,C 0.000} C_DIS
LIN {X 23.113,Y -21.308,Z -43.308,A -90.000,B 90.000,C 0.000} C_DIS
LIN {X 24.563,Y -21.308,Z -43.120,A -90.000,B 90.000,C 0.000} C_DIS
LIN {X 24.951,Y -21.308,Z -43.068,A -90.000,B 90.000,C 0.000} C_DIS
LIN {X 25.986,Y -21.308,Z -42.858,A -90.000,B 90.000,C 0.000} C_DIS
LIN {X 27.080,Y -21.308,Z -42.621,A -90.000,B 90.000,C 0.000} C_DIS
LIN {X 29.127,Y -21.308,Z -42.046,A -90.000,B 90.000,C 0.000} C_DIS
LIN {X 30.521,Y -21.308,Z -41.604,A -90.000,B 90.000,C 0.000} C_DIS
LIN {X 31.527,Y -21.308,Z -41.318,A -90.000,B 90.000,C 0.000} C_DIS
LIN {X 32.010,Y -21.308,Z -41.160,A -90.000,B 90.000,C 0.000} C_DIS
LIN {X 32.404,Y -21.308,Z -41.038,A -90.000,B 90.000,C 0.000} C_DIS
LIN {X 33.016,Y -21.308,Z -40.857,A -90.000,B 90.000,C 0.000} C_DIS
LIN {X 33.779,Y -21.308,Z -40.642,A -90.000,B 90.000,C 0.000} C_DIS
LIN {X 34.566,Y -21.308,Z -40.465,A -90.000,B 90.000,C 0.000} C_DIS
LIN {X 35.182,Y -21.308,Z -40.306,A -90.000,B 90.000,C 0.000} C_DIS
LIN {X 35.761,Y -21.308,Z -40.171,A -90.000,B 90.000,C 0.000} C_DIS
LIN {X 36.808,Y -21.308,Z -39.968,A -90.000,B 90.000,C 0.000} C_DIS
LIN {X 37.211,Y -21.308,Z -39.897,A -90.000,B 90.000,C 0.000} C_DIS
LIN {X 37.756,Y -21.308,Z -39.826,A -90.000,B 90.000,C 0.000} C_DIS
LIN {X 37.897,Y -21.308,Z -39.809,A -90.000,B 90.000,C 0.000} C_DIS
LIN {X 39.241,Y -21.308,Z -39.667,A -90.000,B 90.000,C 0.000} C_DIS
LIN {X 39.706,Y -21.308,Z -39.626,A -90.000,B 90.000,C 0.000} C_DIS
LIN {X 41.257,Y -21.308,Z -39.593,A -90.000,B 90.000,C 0.000} C_DIS
LIN {X 41.772,Y -21.308,Z -39.604,A -90.000,B 90.000,C 0.000} C_DIS
LIN {X 42.247,Y -21.308,Z -39.627,A -90.000,B 90.000,C 0.000} C_DIS
LIN {X 42.838,Y -21.308,Z -39.676,A -90.000,B 90.000,C 0.000} C_DIS
LIN {X 43.812,Y -21.308,Z -39.783,A -90.000,B 90.000,C 0.000} C_DIS
LIN {X 44.323,Y -21.308,Z -39.847,A -90.000,B 90.000,C 0.000} C_DIS
LIN {X 44.798,Y -21.308,Z -39.930,A -90.000,B 90.000,C 0.000} C_DIS
LIN {X 45.212,Y -21.308,Z -40.007,A -90.000,B 90.000,C 0.000} C_DIS
LIN {X 46.366,Y -21.308,Z -40.300,A -90.000,B 90.000,C 0.000} C_DIS
LIN {X 46.830,Y -21.308,Z -40.432,A -90.000,B 90.000,C 0.000} C_DIS
LIN {X 48.386,Y -21.308,Z -40.922,A -90.000,B 90.000,C 0.000} C_DIS
LIN {X 48.630,Y -21.308,Z -41.001,A -90.000,B 90.000,C 0.000} C_DIS
LIN {X 49.079,Y -21.308,Z -41.181,A -90.000,B 90.000,C 0.000} C_DIS
LIN {X 49.909,Y -21.308,Z -41.547,A -90.000,B 90.000,C 0.000} C_DIS
LIN {X 51.058,Y -21.308,Z -42.093,A -90.000,B 90.000,C 0.000} C_DIS
LIN {X 51.853,Y -21.308,Z -42.485,A -90.000,B 90.000,C 0.000} C_DIS
LIN {X 52.282,Y -21.308,Z -42.715,A -90.000,B 90.000,C 0.000} C_DIS
LIN {X 54.893,Y -21.308,Z -44.272,A -90.000,B 90.000,C 0.000} C_DIS
LIN {X 55.296,Y -21.308,Z -44.545,A -90.000,B 90.000,C 0.000} C_DIS
LIN {X 56.492,Y -21.308,Z -45.426,A -90.000,B 90.000,C 0.000} C_DIS
LIN {X 57.246,Y -21.308,Z -45.992,A -90.000,B 90.000,C 0.000} C_DIS
LIN {X 57.589,Y -21.308,Z -46.239,A -90.000,B 90.000,C 0.000} C_DIS
LIN {X 57.963,Y -21.308,Z -46.554,A -90.000,B 90.000,C 0.000} C_DIS
LIN {X 59.523,Y -21.308,Z -47.890,A -90.000,B 90.000,C 0.000} C_DIS
LIN {X 60.020,Y -21.308,Z -48.325,A -90.000,B 90.000,C 0.000} C_DIS
LIN {X 61.895,Y -21.308,Z -50.056,A -90.000,B 90.000,C 0.000} C_DIS
LIN {X 62.447,Y -21.308,Z -50.533,A -90.000,B 90.000,C 0.000} C_DIS
LIN {X 63.559,Y -21.308,Z -51.540,A -90.000,B 90.000,C 0.000} C_DIS
LIN {X 64.754,Y -21.308,Z -52.467,A -90.000,B 90.000,C 0.000} C_DIS
LIN {X 65.201,Y -21.308,Z -52.828,A -90.000,B 90.000,C 0.000} C_DIS
LIN {X 66.418,Y -21.308,Z -53.618,A -90.000,B 90.000,C 0.000} C_DIS
LIN {X 66.971,Y -21.308,Z -53.957,A -90.000,B 90.000,C 0.000} C_DIS
LIN {X 68.245,Y -21.308,Z -54.717,A -90.000,B 90.000,C 0.000} C_DIS
LIN {X 69.164,Y -21.308,Z -55.250,A -90.000,B 90.000,C 0.000} C_DIS
LIN {X 70.153,Y -21.308,Z -55.847,A -90.000,B 90.000,C 0.000} C_DIS
LIN {X 71.301,Y -21.308,Z -56.531,A -90.000,B 90.000,C 0.000} C_DIS
LIN {X 71.703,Y -21.308,Z -56.798,A -90.000,B 90.000,C 0.000} C_DIS
LIN {X 72.358,Y -21.308,Z -57.238,A -90.000,B 90.000,C 0.000} C_DIS
LIN {X 73.667,Y -21.308,Z -58.106,A -90.000,B 90.000,C 0.000} C_DIS
LIN {X 74.716,Y -21.308,Z -58.956,A -90.000,B 90.000,C 0.000} C_DIS
LIN {X 75.681,Y -21.308,Z -59.755,A -90.000,B 90.000,C 0.000} C_DIS
LIN {X 77.039,Y -21.308,Z -61.068,A -90.000,B 90.000,C 0.000} C_DIS
LIN {X 77.433,Y -21.308,Z -61.461,A -90.000,B 90.000,C 0.000} C_DIS
LIN {X 78.478,Y -21.308,Z -62.635,A -90.000,B 90.000,C 0.000} C_DIS
LIN {X 78.670,Y -21.308,Z -62.865,A -90.000,B 90.000,C 0.000} C_DIS
LIN {X 78.979,Y -21.308,Z -63.248,A -90.000,B 90.000,C 0.000} C_DIS
LIN {X 79.119,Y -21.308,Z -63.424,A -90.000,B 90.000,C 0.000} C_DIS
LIN {X 79.746,Y -21.308,Z -61.546,A -90.000,B 90.000,C 0.000} C_DIS
LIN {X 79.783,Y -21.308,Z -61.448,A -90.000,B 90.000,C 0.000} C_DIS
LIN {X 80.316,Y -21.308,Z -59.745,A -90.000,B 90.000,C 0.000} C_DIS
LIN {X 80.461,Y -21.308,Z -59.314,A -90.000,B 90.000,C 0.000} C_DIS
LIN {X 81.203,Y -21.308,Z -57.299,A -90.000,B 90.000,C 0.000} C_DIS
LIN {X 81.700,Y -21.308,Z -56.182,A -90.000,B 90.000,C 0.000} C_DIS
LIN {X 82.139,Y -21.308,Z -55.098,A -90.000,B 90.000,C 0.000} C_DIS
LIN {X 82.335,Y -21.308,Z -54.666,A -90.000,B 90.000,C 0.000} C_DIS
LIN {X 83.331,Y -21.308,Z -52.811,A -90.000,B 90.000,C 0.000} C_DIS
LIN {X 83.577,Y -21.308,Z -52.389,A -90.000,B 90.000,C 0.000} C_DIS
LIN {X 84.746,Y -21.308,Z -50.672,A -90.000,B 90.000,C 0.000} C_DIS
LIN {X 85.025,Y -21.308,Z -50.291,A -90.000,B 90.000,C 0.000} C_DIS
LIN {X 86.337,Y -21.308,Z -48.714,A -90.000,B 90.000,C 0.000} C_DIS
LIN {X 86.388,Y -21.308,Z -48.657,A -90.000,B 90.000,C 0.000} C_DIS
LIN {X 86.664,Y -21.308,Z -48.352,A -90.000,B 90.000,C 0.000} C_DIS
LIN {X 88.117,Y -21.308,Z -46.880,A -90.000,B 90.000,C 0.000} C_DIS
LIN {X 88.539,Y -21.308,Z -46.500,A -90.000,B 90.000,C 0.000} C_DIS
LIN {X 90.061,Y -21.308,Z -45.164,A -90.000,B 90.000,C 0.000} C_DIS
LIN {X 91.734,Y -21.308,Z -43.863,A -90.000,B 90.000,C 0.000} C_DIS
LIN {X 92.110,Y -21.308,Z -43.588,A -90.000,B 90.000,C 0.000} C_DIS
LIN {X 93.780,Y -21.308,Z -42.419,A -90.000,B 90.000,C 0.000} C_DIS
LIN {X 95.441,Y -21.308,Z -41.368,A -90.000,B 90.000,C 0.000} C_DIS
LIN {X 95.927,Y -21.308,Z -41.085,A -90.000,B 90.000,C 0.000} C_DIS
LIN {X 97.376,Y -21.308,Z -40.260,A -90.000,B 90.000,C 0.000} C_DIS
LIN {X 98.805,Y -21.308,Z -39.523,A -90.000,B 90.000,C 0.000} C_DIS
LIN {X 100.266,Y -21.308,Z -38.830,A -90.000,B 90.000,C 0.000} C_DIS
LIN {X 102.132,Y -21.308,Z -37.985,A -90.000,B 90.000,C 0.000} C_DIS
LIN {X 103.331,Y -21.308,Z -37.449,A -90.000,B 90.000,C 0.000} C_DIS
LIN {X 104.475,Y -21.308,Z -36.943,A -90.000,B 90.000,C 0.000} C_DIS
LIN {X 105.369,Y -21.308,Z -36.566,A -90.000,B 90.000,C 0.000} C_DIS
LIN {X 106.892,Y -21.308,Z -35.961,A -90.000,B 90.000,C 0.000} C_DIS
LIN {X 107.415,Y -21.308,Z -35.762,A -90.000,B 90.000,C 0.000} C_DIS
LIN {X 107.855,Y -21.308,Z -35.604,A -90.000,B 90.000,C 0.000} C_DIS
LIN {X 108.317,Y -21.308,Z -35.448,A -90.000,B 90.000,C 0.000} C_DIS
LIN {X 108.745,Y -21.308,Z -35.333,A -90.000,B 90.000,C 0.000} C_DIS
LIN {X 109.221,Y -21.308,Z -35.225,A -90.000,B 90.000,C 0.000} C_DIS
LIN {X 109.669,Y -21.308,Z -35.166,A -90.000,B 90.000,C 0.000} C_DIS
LIN {X 110.108,Y -21.308,Z -35.113,A -90.000,B 90.000,C 0.000} C_DIS
LIN {X 110.596,Y -21.308,Z -35.105,A -90.000,B 90.000,C 0.000} C_DIS
LIN {X 110.949,Y -21.308,Z -35.117,A -90.000,B 90.000,C 0.000} C_DIS
LIN {X 111.435,Y -21.308,Z -35.158,A -90.000,B 90.000,C 0.000} C_DIS
LIN {X 112.068,Y -21.308,Z -35.277,A -90.000,B 90.000,C 0.000} C_DIS
LIN {X 112.405,Y -21.308,Z -35.362,A -90.000,B 90.000,C 0.000} C_DIS
LIN {X 112.592,Y -21.308,Z -35.418,A -90.000,B 90.000,C 0.000} C_DIS
LIN {X 112.946,Y -21.308,Z -35.525,A -90.000,B 90.000,C 0.000} C_DIS
LIN {X 113.055,Y -21.308,Z -35.560,A -90.000,B 90.000,C 0.000} C_DIS
LIN {X 113.505,Y -21.308,Z -35.746,A -90.000,B 90.000,C 0.000} C_DIS
LIN {X 113.979,Y -21.308,Z -35.973,A -90.000,B 90.000,C 0.000} C_DIS
LIN {X 114.422,Y -21.308,Z -36.212,A -90.000,B 90.000,C 0.000} C_DIS
LIN {X 114.540,Y -21.308,Z -36.286,A -90.000,B 90.000,C 0.000} C_DIS
LIN {X 114.954,Y -21.308,Z -36.568,A -90.000,B 90.000,C 0.000} C_DIS
LIN {X 115.050,Y -21.308,Z -36.644,A -90.000,B 90.000,C 0.000} C_DIS
LIN {X 115.432,Y -21.308,Z -36.966,A -90.000,B 90.000,C 0.000} C_DIS
LIN {X 115.513,Y -21.308,Z -37.039,A -90.000,B 90.000,C 0.000} C_DIS
LIN {X 115.945,Y -21.308,Z -37.488,A -90.000,B 90.000,C 0.000} C_DIS
LIN {X 116.082,Y -21.308,Z -37.634,A -90.000,B 90.000,C 0.000} C_DIS
LIN {X 116.439,Y -21.308,Z -38.088,A -90.000,B 90.000,C 0.000} C_DIS
LIN {X 116.700,Y -21.308,Z -38.500,A -90.000,B 90.000,C 0.000} C_DIS
LIN {X 116.931,Y -21.308,Z -38.969,A -90.000,B 90.000,C 0.000} C_DIS
LIN {X 117.060,Y -21.308,Z -39.252,A -90.000,B 90.000,C 0.000} C_DIS
LIN {X 117.107,Y -21.308,Z -39.373,A -90.000,B 90.000,C 0.000} C_DIS
LIN {X 117.260,Y -21.308,Z -39.781,A -90.000,B 90.000,C 0.000} C_DIS
LIN {X 117.392,Y -21.308,Z -40.289,A -90.000,B 90.000,C 0.000} C_DIS
LIN {X 117.462,Y -21.308,Z -40.593,A -90.000,B 90.000,C 0.000} C_DIS
LIN {X 117.542,Y -21.308,Z -41.119,A -90.000,B 90.000,C 0.000} C_DIS
LIN {X 117.593,Y -21.308,Z -41.494,A -90.000,B 90.000,C 0.000} C_DIS
LIN {X 117.630,Y -21.308,Z -41.874,A -90.000,B 90.000,C 0.000} C_DIS
LIN {X 117.657,Y -21.308,Z -42.395,A -90.000,B 90.000,C 0.000} C_DIS
LIN {X 117.668,Y -21.308,Z -42.701,A -90.000,B 90.000,C 0.000} C_DIS
LIN {X 117.664,Y -21.308,Z -42.876,A -90.000,B 90.000,C 0.000} C_DIS
LIN {X 117.651,Y -21.308,Z -43.202,A -90.000,B 90.000,C 0.000} C_DIS
LIN {X 117.606,Y -21.308,Z -43.732,A -90.000,B 90.000,C 0.000} C_DIS
LIN {X 117.567,Y -21.308,Z -44.117,A -90.000,B 90.000,C 0.000} C_DIS
LIN {X 117.489,Y -21.308,Z -44.635,A -90.000,B 90.000,C 0.000} C_DIS
LIN {X 117.399,Y -21.308,Z -45.114,A -90.000,B 90.000,C 0.000} C_DIS
LIN {X 117.260,Y -21.308,Z -45.739,A -90.000,B 90.000,C 0.000} C_DIS
LIN {X 117.204,Y -21.308,Z -45.929,A -90.000,B 90.000,C 0.000} C_DIS
LIN {X 116.900,Y -21.308,Z -46.938,A -90.000,B 90.000,C 0.000} C_DIS
LIN {X 116.541,Y -21.308,Z -47.870,A -90.000,B 90.000,C 0.000} C_DIS
LIN {X 116.372,Y -21.308,Z -48.278,A -90.000,B 90.000,C 0.000} C_DIS
LIN {X 115.873,Y -21.308,Z -49.350,A -90.000,B 90.000,C 0.000} C_DIS
LIN {X 115.217,Y -21.308,Z -50.661,A -90.000,B 90.000,C 0.000} C_DIS
LIN {X 114.622,Y -21.308,Z -51.838,A -90.000,B 90.000,C 0.000} C_DIS
LIN {X 113.941,Y -21.308,Z -53.229,A -90.000,B 90.000,C 0.000} C_DIS
LIN {X 113.276,Y -21.308,Z -54.687,A -90.000,B 90.000,C 0.000} C_DIS
LIN {X 112.799,Y -21.308,Z -55.830,A -90.000,B 90.000,C 0.000} C_DIS
LIN {X 112.213,Y -21.308,Z -57.388,A -90.000,B 90.000,C 0.000} C_DIS
LIN {X 111.674,Y -21.308,Z -59.009,A -90.000,B 90.000,C 0.000} C_DIS
LIN {X 111.260,Y -21.308,Z -60.445,A -90.000,B 90.000,C 0.000} C_DIS
LIN {X 110.736,Y -21.308,Z -62.369,A -90.000,B 90.000,C 0.000} C_DIS
LIN {X 110.149,Y -21.308,Z -64.450,A -90.000,B 90.000,C 0.000} C_DIS
LIN {X 110.021,Y -21.308,Z -64.879,A -90.000,B 90.000,C 0.000} C_DIS
LIN {X 109.345,Y -21.308,Z -67.050,A -90.000,B 90.000,C 0.000} C_DIS
LIN {X 108.519,Y -21.308,Z -69.358,A -90.000,B 90.000,C 0.000} C_DIS
LIN {X 107.575,Y -21.308,Z -71.732,A -90.000,B 90.000,C 0.000} C_DIS
LIN {X 107.403,Y -21.308,Z -72.150,A -90.000,B 90.000,C 0.000} C_DIS
LIN {X 106.414,Y -21.308,Z -74.420,A -90.000,B 90.000,C 0.000} C_DIS
LIN {X 105.411,Y -21.308,Z -76.516,A -90.000,B 90.000,C 0.000} C_DIS
LIN {X 104.209,Y -21.308,Z -78.763,A -90.000,B 90.000,C 0.000} C_DIS
LIN {X 103.918,Y -21.308,Z -79.266,A -90.000,B 90.000,C 0.000} C_DIS
LIN {X 103.058,Y -21.308,Z -80.726,A -90.000,B 90.000,C 0.000} C_DIS
LIN {X 102.198,Y -21.308,Z -82.078,A -90.000,B 90.000,C 0.000} C_DIS
LIN {X 100.858,Y -21.308,Z -84.085,A -90.000,B 90.000,C 0.000} C_DIS
LIN {X 99.737,Y -21.308,Z -85.762,A -90.000,B 90.000,C 0.000} C_DIS
LIN {X 99.861,Y -21.308,Z -87.356,A -90.000,B 90.000,C 0.000} C_DIS
LIN {X 100.041,Y -21.308,Z -89.925,A -90.000,B 90.000,C 0.000} C_DIS
LIN {X 100.046,Y -21.308,Z -89.994,A -90.000,B 90.000,C 0.000} C_DIS
LIN {X 100.213,Y -21.308,Z -90.848,A -90.000,B 90.000,C 0.000} C_DIS
LIN {X 100.318,Y -21.308,Z -91.520,A -90.000,B 90.000,C 0.000} C_DIS
LIN {X 100.421,Y -21.308,Z -92.375,A -90.000,B 90.000,C 0.000} C_DIS
LIN {X 100.448,Y -21.308,Z -92.525,A -90.000,B 90.000,C 0.000} C_DIS
LIN {X 100.523,Y -21.308,Z -93.006,A -90.000,B 90.000,C 0.000} C_DIS
LIN {X 100.548,Y -21.308,Z -93.492,A -90.000,B 90.000,C 0.000} C_DIS
LIN {X 100.554,Y -21.308,Z -93.759,A -90.000,B 90.000,C 0.000} C_DIS
LIN {X 100.618,Y -21.308,Z -94.493,A -90.000,B 90.000,C 0.000} C_DIS
LIN {X 100.641,Y -21.308,Z -94.947,A -90.000,B 90.000,C 0.000} C_DIS
LIN {X 100.639,Y -21.308,Z -95.024,A -90.000,B 90.000,C 0.000} C_DIS
LIN {X 100.647,Y -21.308,Z -95.315,A -90.000,B 90.000,C 0.000} C_DIS
LIN {X 100.658,Y -21.308,Z -95.921,A -90.000,B 90.000,C 0.000} C_DIS
LIN {X 100.674,Y -21.308,Z -96.224,A -90.000,B 90.000,C 0.000} C_DIS
LIN {X 100.672,Y -21.308,Z -97.155,A -90.000,B 90.000,C 0.000} C_DIS
LIN {X 100.688,Y -21.308,Z -97.358,A -90.000,B 90.000,C 0.000} C_DIS
LIN {X 100.728,Y -21.308,Z -98.111,A -90.000,B 90.000,C 0.000} C_DIS
LIN {X 100.732,Y -21.308,Z -98.811,A -90.000,B 90.000,C 0.000} C_DIS
LIN {X 100.756,Y -21.308,Z -99.073,A -90.000,B 90.000,C 0.000} C_DIS
LIN {X 100.781,Y -21.308,Z -99.549,A -90.000,B 90.000,C 0.000} C_DIS
LIN {X 100.788,Y -21.308,Z -100.316,A -90.000,B 90.000,C 0.000} C_DIS
LIN {X 100.811,Y -21.308,Z -100.538,A -90.000,B 90.000,C 0.000} C_DIS
LIN {X 100.836,Y -21.308,Z -101.014,A -90.000,B 90.000,C 0.000} C_DIS
LIN {X 100.855,Y -21.308,Z -101.837,A -90.000,B 90.000,C 0.000} C_DIS
LIN {X 100.903,Y -21.308,Z -102.292,A -90.000,B 90.000,C 0.000} C_DIS
LIN {X 100.928,Y -21.308,Z -102.758,A -90.000,B 90.000,C 0.000} C_DIS
LIN {X 100.952,Y -21.308,Z -103.221,A -90.000,B 90.000,C 0.000} C_DIS
LIN {X 101.033,Y -21.308,Z -103.993,A -90.000,B 90.000,C 0.000} C_DIS
LIN {X 101.113,Y -21.308,Z -104.565,A -90.000,B 90.000,C 0.000} C_DIS
LIN {X 101.190,Y -21.308,Z -105.068,A -90.000,B 90.000,C 0.000} C_DIS
LIN {X 101.282,Y -21.308,Z -105.614,A -90.000,B 90.000,C 0.000} C_DIS
LIN {X 101.421,Y -21.308,Z -106.435,A -90.000,B 90.000,C 0.000} C_DIS
LIN {X 101.519,Y -21.308,Z -107.043,A -90.000,B 90.000,C 0.000} C_DIS
LIN {X 101.645,Y -21.308,Z -107.874,A -90.000,B 90.000,C 0.000} C_DIS
LIN {X 101.671,Y -21.308,Z -108.050,A -90.000,B 90.000,C 0.000} C_DIS
LIN {X 101.764,Y -21.308,Z -108.793,A -90.000,B 90.000,C 0.000} C_DIS
LIN {X 101.820,Y -21.308,Z -109.211,A -90.000,B 90.000,C 0.000} C_DIS
LIN {X 101.936,Y -21.308,Z -110.227,A -90.000,B 90.000,C 0.000} C_DIS
LIN {X 102.000,Y -21.308,Z -110.740,A -90.000,B 90.000,C 0.000} C_DIS
LIN {X 102.144,Y -21.308,Z -112.050,A -90.000,B 90.000,C 0.000} C_DIS
LIN {X 102.208,Y -21.308,Z -112.580,A -90.000,B 90.000,C 0.000} C_DIS
LIN {X 102.382,Y -21.308,Z -114.138,A -90.000,B 90.000,C 0.000} C_DIS
LIN {X 102.511,Y -21.308,Z -115.194,A -90.000,B 90.000,C 0.000} C_DIS
LIN {X 102.761,Y -21.308,Z -117.353,A -90.000,B 90.000,C 0.000} C_DIS
LIN {X 103.008,Y -21.308,Z -119.583,A -90.000,B 90.000,C 0.000} C_DIS
LIN {X 103.090,Y -21.308,Z -120.387,A -90.000,B 90.000,C 0.000} C_DIS
LIN {X 103.225,Y -21.308,Z -121.748,A -90.000,B 90.000,C 0.000} C_DIS
LIN {X 103.306,Y -21.308,Z -122.667,A -90.000,B 90.000,C 0.000} C_DIS
LIN {X 103.429,Y -21.308,Z -124.198,A -90.000,B 90.000,C 0.000} C_DIS
LIN {X 103.526,Y -21.308,Z -126.043,A -90.000,B 90.000,C 0.000} C_DIS
LIN {X 103.560,Y -21.308,Z -126.586,A -90.000,B 90.000,C 0.000} C_DIS
LIN {X 103.585,Y -21.308,Z -127.041,A -90.000,B 90.000,C 0.000} C_DIS
LIN {X 103.627,Y -21.308,Z -128.934,A -90.000,B 90.000,C 0.000} C_DIS
LIN {X 103.646,Y -21.308,Z -129.477,A -90.000,B 90.000,C 0.000} C_DIS
LIN {X 103.635,Y -21.308,Z -131.610,A -90.000,B 90.000,C 0.000} C_DIS
LIN {X 103.638,Y -21.308,Z -132.073,A -90.000,B 90.000,C 0.000} C_DIS
LIN {X 103.637,Y -21.308,Z -132.183,A -90.000,B 90.000,C 0.000} C_DIS
LIN {X 103.572,Y -21.308,Z -134.627,A -90.000,B 90.000,C 0.000} C_DIS
LIN {X 103.565,Y -21.308,Z -135.047,A -90.000,B 90.000,C 0.000} C_DIS
LIN {X 103.549,Y -21.308,Z -135.492,A -90.000,B 90.000,C 0.000} C_DIS
LIN {X 103.428,Y -21.308,Z -138.376,A -90.000,B 90.000,C 0.000} C_DIS
LIN {X 103.352,Y -21.308,Z -139.990,A -90.000,B 90.000,C 0.000} C_DIS
LIN {X 103.249,Y -21.308,Z -141.903,A -90.000,B 90.000,C 0.000} C_DIS
LIN {X 103.151,Y -21.308,Z -143.612,A -90.000,B 90.000,C 0.000} C_DIS
LIN {X 103.026,Y -21.308,Z -145.605,A -90.000,B 90.000,C 0.000} C_DIS
LIN {X 102.905,Y -21.308,Z -147.473,A -90.000,B 90.000,C 0.000} C_DIS
LIN {X 102.770,Y -21.308,Z -149.384,A -90.000,B 90.000,C 0.000} C_DIS
LIN {X 102.642,Y -21.308,Z -151.025,A -90.000,B 90.000,C 0.000} C_DIS
LIN {X 102.493,Y -21.308,Z -153.139,A -90.000,B 90.000,C 0.000} C_DIS
LIN {X 102.381,Y -21.308,Z -154.464,A -90.000,B 90.000,C 0.000} C_DIS
LIN {X 102.201,Y -21.308,Z -156.877,A -90.000,B 90.000,C 0.000} C_DIS
LIN {X 102.115,Y -21.308,Z -157.832,A -90.000,B 90.000,C 0.000} C_DIS
LIN {X 101.899,Y -21.308,Z -160.595,A -90.000,B 90.000,C 0.000} C_DIS
LIN {X 101.854,Y -21.308,Z -161.070,A -90.000,B 90.000,C 0.000} C_DIS
LIN {X 101.595,Y -21.308,Z -164.284,A -90.000,B 90.000,C 0.000} C_DIS
LIN {X 101.465,Y -21.308,Z -165.828,A -90.000,B 90.000,C 0.000} C_DIS
LIN {X 101.266,Y -21.308,Z -168.014,A -90.000,B 90.000,C 0.000} C_DIS
LIN {X 100.914,Y -21.308,Z -171.688,A -90.000,B 90.000,C 0.000} C_DIS
LIN {X 100.553,Y -21.308,Z -175.231,A -90.000,B 90.000,C 0.000} C_DIS
LIN {X 100.494,Y -21.308,Z -175.773,A -90.000,B 90.000,C 0.000} C_DIS
LIN {X 100.196,Y -21.308,Z -178.377,A -90.000,B 90.000,C 0.000} C_DIS
LIN {X 99.833,Y -21.308,Z -181.228,A -90.000,B 90.000,C 0.000} C_DIS
LIN {X 99.473,Y -21.308,Z -183.855,A -90.000,B 90.000,C 0.000} C_DIS
LIN {X 99.362,Y -21.308,Z -184.639,A -90.000,B 90.000,C 0.000} C_DIS
LIN {X 98.972,Y -21.308,Z -187.361,A -90.000,B 90.000,C 0.000} C_DIS
LIN {X 98.774,Y -21.308,Z -188.724,A -90.000,B 90.000,C 0.000} C_DIS
LIN {X 98.597,Y -21.308,Z -190.008,A -90.000,B 90.000,C 0.000} C_DIS
LIN {X 98.444,Y -21.308,Z -191.104,A -90.000,B 90.000,C 0.000} C_DIS
LIN {X 98.196,Y -21.308,Z -192.748,A -90.000,B 90.000,C 0.000} C_DIS
LIN {X 98.054,Y -21.308,Z -193.666,A -90.000,B 90.000,C 0.000} C_DIS
LIN {X 97.674,Y -21.308,Z -195.833,A -90.000,B 90.000,C 0.000} C_DIS
LIN {X 97.511,Y -21.308,Z -196.714,A -90.000,B 90.000,C 0.000} C_DIS
LIN {X 97.445,Y -21.308,Z -197.054,A -90.000,B 90.000,C 0.000} C_DIS
LIN {X 96.854,Y -21.308,Z -199.954,A -90.000,B 90.000,C 0.000} C_DIS
LIN {X 96.721,Y -21.308,Z -200.570,A -90.000,B 90.000,C 0.000} C_DIS
LIN {X 95.807,Y -21.308,Z -204.533,A -90.000,B 90.000,C 0.000} C_DIS
LIN {X 95.724,Y -21.308,Z -204.878,A -90.000,B 90.000,C 0.000} C_DIS
LIN {X 94.532,Y -21.308,Z -209.736,A -90.000,B 90.000,C 0.000} C_DIS
LIN {X 94.209,Y -21.308,Z -211.007,A -90.000,B 90.000,C 0.000} C_DIS
LIN {X 93.186,Y -21.308,Z -214.997,A -90.000,B 90.000,C 0.000} C_DIS
LIN {X 93.115,Y -21.308,Z -215.282,A -90.000,B 90.000,C 0.000} C_DIS
LIN {X 91.766,Y -21.308,Z -220.467,A -90.000,B 90.000,C 0.000} C_DIS
LIN {X 90.586,Y -21.308,Z -224.974,A -90.000,B 90.000,C 0.000} C_DIS
LIN {X 90.336,Y -21.308,Z -225.952,A -90.000,B 90.000,C 0.000} C_DIS
LIN {X 88.794,Y -21.308,Z -231.545,A -90.000,B 90.000,C 0.000} C_DIS
LIN {X 87.569,Y -21.308,Z -235.603,A -90.000,B 90.000,C 0.000} C_DIS
LIN {X 87.046,Y -21.308,Z -237.337,A -90.000,B 90.000,C 0.000} C_DIS
LIN {X 86.911,Y -21.308,Z -237.772,A -90.000,B 90.000,C 0.000} C_DIS
LIN {X 85.571,Y -21.308,Z -241.745,A -90.000,B 90.000,C 0.000} C_DIS
LIN {X 84.966,Y -21.308,Z -243.561,A -90.000,B 90.000,C 0.000} C_DIS
LIN {X 84.966,Y -60.000,Z -243.561,A -90.000,B 90.000,C 0.000} C_DIS
LIN {X 100.049,Y -60.000,Z -89.971,A -90.000,B 90.000,C 0.000} C_DIS
LIN {X 100.049,Y -19.308,Z -89.971,A -90.000,B 90.000,C 0.000} C_DIS
LIN {X 100.370,Y -19.311,Z -91.184,A -90.000,B 90.000,C 0.000} C_DIS
LIN {X 100.503,Y -19.315,Z -91.698,A -90.000,B 90.000,C 0.000} C_DIS
LIN {X 100.648,Y -19.318,Z -92.535,A -90.000,B 90.000,C 0.000} C_DIS
LIN {X 100.763,Y -19.323,Z -93.031,A -90.000,B 90.000,C 0.000} C_DIS
LIN {X 100.834,Y -19.329,Z -93.495,A -90.000,B 90.000,C 0.000} C_DIS
LIN {X 100.875,Y -19.331,Z -94.001,A -90.000,B 90.000,C 0.000} C_DIS
LIN {X 100.939,Y -19.335,Z -94.444,A -90.000,B 90.000,C 0.000} C_DIS
LIN {X 100.992,Y -19.341,Z -94.807,A -90.000,B 90.000,C 0.000} C_DIS
LIN {X 101.011,Y -19.343,Z -95.164,A -90.000,B 90.000,C 0.000} C_DIS
LIN {X 101.085,Y -19.353,Z -96.020,A -90.000,B 90.000,C 0.000} C_DIS
LIN {X 101.104,Y -19.355,Z -96.412,A -90.000,B 90.000,C 0.000} C_DIS
LIN {X 101.155,Y -19.366,Z -97.195,A -90.000,B 90.000,C 0.000} C_DIS
LIN {X 101.166,Y -19.367,Z -97.318,A -90.000,B 90.000,C 0.000} C_DIS
LIN {X 101.182,Y -19.369,Z -97.446,A -90.000,B 90.000,C 0.000} C_DIS
LIN {X 101.210,Y -19.371,Z -97.821,A -90.000,B 90.000,C 0.000} C_DIS
LIN {X 101.231,Y -19.373,Z -98.097,A -90.000,B 90.000,C 0.000} C_DIS
LIN {X 101.268,Y -19.382,Z -98.616,A -90.000,B 90.000,C 0.000} C_DIS
LIN {X 101.289,Y -19.387,Z -98.761,A -90.000,B 90.000,C 0.000} C_DIS
LIN {X 101.312,Y -19.388,Z -99.044,A -90.000,B 90.000,C 0.000} C_DIS
LIN {X 101.360,Y -19.394,Z -99.633,A -90.000,B 90.000,C 0.000} C_DIS
LIN {X 101.398,Y -19.404,Z -100.109,A -90.000,B 90.000,C 0.000} C_DIS
LIN {X 101.403,Y -19.406,Z -100.144,A -90.000,B 90.000,C 0.000} C_DIS
LIN {X 101.415,Y -19.409,Z -100.281,A -90.000,B 90.000,C 0.000} C_DIS
LIN {X 101.448,Y -19.411,Z -100.635,A -90.000,B 90.000,C 0.000} C_DIS
LIN {X 101.479,Y -19.416,Z -100.960,A -90.000,B 90.000,C 0.000} C_DIS
LIN {X 101.541,Y -19.431,Z -101.635,A -90.000,B 90.000,C 0.000} C_DIS
LIN {X 101.545,Y -19.432,Z -101.726,A -90.000,B 90.000,C 0.000} C_DIS
LIN {X 101.555,Y -19.435,Z -101.800,A -90.000,B 90.000,C 0.000} C_DIS
LIN {X 101.578,Y -19.437,Z -101.959,A -90.000,B 90.000,C 0.000} C_DIS
LIN {X 101.617,Y -19.439,Z -102.324,A -90.000,B 90.000,C 0.000} C_DIS
LIN {X 101.702,Y -19.455,Z -103.172,A -90.000,B 90.000,C 0.000} C_DIS
LIN {X 101.718,Y -19.455,Z -103.318,A -90.000,B 90.000,C 0.000} C_DIS
LIN {X 101.809,Y -19.461,Z -104.017,A -90.000,B 90.000,C 0.000} C_DIS
LIN {X 101.864,Y -19.460,Z -104.421,A -90.000,B 90.000,C 0.000} C_DIS
LIN {X 102.006,Y -19.459,Z -105.329,A -90.000,B 90.000,C 0.000} C_DIS
LIN {X 102.233,Y -19.454,Z -106.760,A -90.000,B 90.000,C 0.000} C_DIS
LIN {X 102.372,Y -19.454,Z -107.673,A -90.000,B 90.000,C 0.000} C_DIS
LIN {X 102.455,Y -19.455,Z -108.257,A -90.000,B 90.000,C 0.000} C_DIS
LIN {X 102.544,Y -19.458,Z -108.902,A -90.000,B 90.000,C 0.000} C_DIS
LIN {X 102.678,Y -19.464,Z -109.907,A -90.000,B 90.000,C 0.000} C_DIS
LIN {X 102.805,Y -19.468,Z -110.902,A -90.000,B 90.000,C 0.000} C_DIS
LIN {X 102.940,Y -19.475,Z -111.981,A -90.000,B 90.000,C 0.000} C_DIS
LIN {X 103.004,Y -19.475,Z -112.492,A -90.000,B 90.000,C 0.000} C_DIS
LIN {X 103.195,Y -19.484,Z -114.043,A -90.000,B 90.000,C 0.000} C_DIS
LIN {X 103.324,Y -19.484,Z -115.099,A -90.000,B 90.000,C 0.000} C_DIS
LIN {X 103.526,Y -19.488,Z -116.755,A -90.000,B 90.000,C 0.000} C_DIS
LIN {X 103.715,Y -19.490,Z -118.396,A -90.000,B 90.000,C 0.000} C_DIS
LIN {X 103.816,Y -19.493,Z -119.256,A -90.000,B 90.000,C 0.000} C_DIS
LIN {X 103.969,Y -19.494,Z -120.728,A -90.000,B 90.000,C 0.000} C_DIS
LIN {X 104.071,Y -19.498,Z -121.676,A -90.000,B 90.000,C 0.000} C_DIS
LIN {X 104.195,Y -19.500,Z -123.070,A -90.000,B 90.000,C 0.000} C_DIS
LIN {X 104.292,Y -19.505,Z -124.164,A -90.000,B 90.000,C 0.000} C_DIS
LIN {X 104.429,Y -19.515,Z -126.286,A -90.000,B 90.000,C 0.000} C_DIS
LIN {X 104.446,Y -19.516,Z -126.545,A -90.000,B 90.000,C 0.000} C_DIS
LIN {X 104.472,Y -19.516,Z -127.030,A -90.000,B 90.000,C 0.000} C_DIS
LIN {X 104.538,Y -19.528,Z -128.908,A -90.000,B 90.000,C 0.000} C_DIS
LIN {X 104.561,Y -19.530,Z -129.482,A -90.000,B 90.000,C 0.000} C_DIS
LIN {X 104.574,Y -19.542,Z -131.331,A -90.000,B 90.000,C 0.000} C_DIS
LIN {X 104.584,Y -19.546,Z -132.068,A -90.000,B 90.000,C 0.000} C_DIS
LIN {X 104.548,Y -19.557,Z -134.274,A -90.000,B 90.000,C 0.000} C_DIS
LIN {X 104.541,Y -19.562,Z -134.964,A -90.000,B 90.000,C 0.000} C_DIS
LIN {X 104.520,Y -19.564,Z -135.673,A -90.000,B 90.000,C 0.000} C_DIS
LIN {X 104.420,Y -19.575,Z -138.502,A -90.000,B 90.000,C 0.000} C_DIS
LIN {X 104.374,Y -19.577,Z -139.550,A -90.000,B 90.000,C 0.000} C_DIS
LIN {X 104.259,Y -19.583,Z -141.960,A -90.000,B 90.000,C 0.000} C_DIS
LIN {X 104.219,Y -19.585,Z -142.693,A -90.000,B 90.000,C 0.000} C_DIS
LIN {X 104.162,Y -19.585,Z -143.698,A -90.000,B 90.000,C 0.000} C_DIS
LIN {X 104.037,Y -19.590,Z -145.829,A -90.000,B 90.000,C 0.000} C_DIS
LIN {X 103.924,Y -19.589,Z -147.545,A -90.000,B 90.000,C 0.000} C_DIS
LIN {X 103.783,Y -19.593,Z -149.627,A -90.000,B 90.000,C 0.000} C_DIS
LIN {X 103.670,Y -19.595,Z -151.101,A -90.000,B 90.000,C 0.000} C_DIS
LIN {X 103.508,Y -19.591,Z -153.313,A -90.000,B 90.000,C 0.000} C_DIS
LIN {X 103.384,Y -19.592,Z -154.812,A -90.000,B 90.000,C 0.000} C_DIS
LIN {X 103.211,Y -19.586,Z -157.003,A -90.000,B 90.000,C 0.000} C_DIS
LIN {X 103.173,Y -19.588,Z -157.457,A -90.000,B 90.000,C 0.000} C_DIS
LIN {X 103.106,Y -19.587,Z -158.218,A -90.000,B 90.000,C 0.000} C_DIS
LIN {X 102.897,Y -19.578,Z -160.690,A -90.000,B 90.000,C 0.000} C_DIS
LIN {X 102.853,Y -19.580,Z -161.190,A -90.000,B 90.000,C 0.000} C_DIS
LIN {X 102.704,Y -19.572,Z -162.876,A -90.000,B 90.000,C 0.000} C_DIS
LIN {X 102.596,Y -19.567,Z -164.107,A -90.000,B 90.000,C 0.000} C_DIS
LIN {X 102.528,Y -19.565,Z -164.875,A -90.000,B 90.000,C 0.000} C_DIS
LIN {X 102.433,Y -19.561,Z -165.916,A -90.000,B 90.000,C 0.000} C_DIS
LIN {X 102.183,Y -19.561,Z -168.639,A -90.000,B 90.000,C 0.000} C_DIS
LIN {X 101.864,Y -19.560,Z -171.955,A -90.000,B 90.000,C 0.000} C_DIS
LIN {X 101.516,Y -19.557,Z -175.308,A -90.000,B 90.000,C 0.000} C_DIS
LIN {X 101.184,Y -19.557,Z -178.235,A -90.000,B 90.000,C 0.000} C_DIS
LIN {X 101.150,Y -19.555,Z -178.498,A -90.000,B 90.000,C 0.000} C_DIS
LIN {X 100.774,Y -19.554,Z -181.433,A -90.000,B 90.000,C 0.000} C_DIS
LIN {X 100.733,Y -19.553,Z -181.726,A -90.000,B 90.000,C 0.000} C_DIS
LIN {X 100.392,Y -19.544,Z -184.085,A -90.000,B 90.000,C 0.000} C_DIS
LIN {X 99.872,Y -19.528,Z -187.492,A -90.000,B 90.000,C 0.000} C_DIS
LIN {X 99.621,Y -19.520,Z -189.127,A -90.000,B 90.000,C 0.000} C_DIS
LIN {X 99.281,Y -19.508,Z -191.402,A -90.000,B 90.000,C 0.000} C_DIS
LIN {X 99.044,Y -19.502,Z -192.879,A -90.000,B 90.000,C 0.000} C_DIS
LIN {X 98.867,Y -19.500,Z -193.969,A -90.000,B 90.000,C 0.000} C_DIS
LIN {X 98.646,Y -19.499,Z -195.226,A -90.000,B 90.000,C 0.000} C_DIS
LIN {X 98.401,Y -19.496,Z -196.558,A -90.000,B 90.000,C 0.000} C_DIS
LIN {X 98.350,Y -19.496,Z -196.835,A -90.000,B 90.000,C 0.000} C_DIS
LIN {X 98.274,Y -19.496,Z -197.223,A -90.000,B 90.000,C 0.000} C_DIS
LIN {X 98.006,Y -19.501,Z -198.592,A -90.000,B 90.000,C 0.000} C_DIS
LIN {X 97.633,Y -19.497,Z -200.365,A -90.000,B 90.000,C 0.000} C_DIS
LIN {X 97.548,Y -19.498,Z -200.761,A -90.000,B 90.000,C 0.000} C_DIS
LIN {X 97.114,Y -19.510,Z -202.761,A -90.000,B 90.000,C 0.000} C_DIS
LIN {X 96.667,Y -19.506,Z -204.666,A -90.000,B 90.000,C 0.000} C_DIS
LIN {X 96.571,Y -19.508,Z -205.086,A -90.000,B 90.000,C 0.000} C_DIS
LIN {X 95.980,Y -19.526,Z -207.642,A -90.000,B 90.000,C 0.000} C_DIS
LIN {X 95.666,Y -19.530,Z -208.954,A -90.000,B 90.000,C 0.000} C_DIS
LIN {X 95.436,Y -19.529,Z -209.884,A -90.000,B 90.000,C 0.000} C_DIS
LIN {X 94.625,Y -19.553,Z -213.241,A -90.000,B 90.000,C 0.000} C_DIS
LIN {X 94.351,Y -19.562,Z -214.374,A -90.000,B 90.000,C 0.000} C_DIS
LIN {X 94.132,Y -19.562,Z -215.235,A -90.000,B 90.000,C 0.000} C_DIS
LIN {X 94.059,Y -19.562,Z -215.528,A -90.000,B 90.000,C 0.000} C_DIS
LIN {X 92.927,Y -19.588,Z -220.057,A -90.000,B 90.000,C 0.000} C_DIS
LIN {X 92.590,Y -19.589,Z -221.351,A -90.000,B 90.000,C 0.000} C_DIS
LIN {X 91.590,Y -19.598,Z -225.234,A -90.000,B 90.000,C 0.000} C_DIS
LIN {X 91.383,Y -19.598,Z -226.043,A -90.000,B 90.000,C 0.000} C_DIS
LIN {X 91.314,Y -19.597,Z -226.299,A -90.000,B 90.000,C 0.000} C_DIS
LIN {X 89.836,Y -19.598,Z -231.668,A -90.000,B 90.000,C 0.000} C_DIS
LIN {X 89.741,Y -19.596,Z -231.984,A -90.000,B 90.000,C 0.000} C_DIS
LIN {X 88.030,Y -19.594,Z -237.643,A -90.000,B 90.000,C 0.000} C_DIS
LIN {X 87.945,Y -19.594,Z -237.916,A -90.000,B 90.000,C 0.000} C_DIS
LIN {X 87.884,Y -19.592,Z -238.101,A -90.000,B 90.000,C 0.000} C_DIS
LIN {X 86.553,Y -19.598,Z -242.074,A -90.000,B 90.000,C 0.000} C_DIS
LIN {X 86.057,Y -19.597,Z -243.561,A -90.000,B 90.000,C 0.000} C_DIS
LIN {X 86.057,Y -60.000,Z -243.561,A -90.000,B 90.000,C 0.000} C_DIS
LIN {X -107.629,Y -60.000,Z -243.561,A -90.000,B 90.000,C 0.000} C_DIS
LIN {X -107.629,Y -19.815,Z -243.561,A -90.000,B 90.000,C 0.000} C_DIS
LIN {X -107.458,Y -19.698,Z -243.311,A -90.000,B 90.000,C 0.000} C_DIS
LIN {X -107.301,Y -19.633,Z -243.129,A -90.000,B 90.000,C 0.000} C_DIS
LIN {X -107.280,Y -19.626,Z -243.107,A -90.000,B 90.000,C 0.000} C_DIS
LIN {X -107.078,Y -19.582,Z -242.920,A -90.000,B 90.000,C 0.000} C_DIS
LIN {X -106.840,Y -19.567,Z -242.741,A -90.000,B 90.000,C 0.000} C_DIS
LIN {X -103.965,Y -19.580,Z -240.812,A -90.000,B 90.000,C 0.000} C_DIS
LIN {X -101.913,Y -19.598,Z -239.438,A -90.000,B 90.000,C 0.000} C_DIS
LIN {X -96.636,Y -19.668,Z -235.857,A -90.000,B 90.000,C 0.000} C_DIS
LIN {X -95.895,Y -19.677,Z -235.357,A -90.000,B 90.000,C 0.000} C_DIS
LIN {X -92.695,Y -19.725,Z -233.215,A -90.000,B 90.000,C 0.000} C_DIS
LIN {X -88.475,Y -19.794,Z -230.397,A -90.000,B 90.000,C 0.000} C_DIS
LIN {X -87.795,Y -19.803,Z -229.948,A -90.000,B 90.000,C 0.000} C_DIS
LIN {X -84.424,Y -19.857,Z -227.749,A -90.000,B 90.000,C 0.000} C_DIS
LIN {X -82.563,Y -19.891,Z -226.536,A -90.000,B 90.000,C 0.000} C_DIS
LIN {X -80.149,Y -19.929,Z -224.953,A -90.000,B 90.000,C 0.000} C_DIS
LIN {X -79.454,Y -19.935,Z -224.504,A -90.000,B 90.000,C 0.000} C_DIS
LIN {X -74.760,Y -20.004,Z -221.514,A -90.000,B 90.000,C 0.000} C_DIS
LIN {X -73.717,Y -20.019,Z -220.856,A -90.000,B 90.000,C 0.000} C_DIS
LIN {X -72.079,Y -20.031,Z -219.801,A -90.000,B 90.000,C 0.000} C_DIS
LIN {X -66.453,Y -20.073,Z -216.195,A -90.000,B 90.000,C 0.000} C_DIS
LIN {X -64.974,Y -20.089,Z -215.255,A -90.000,B 90.000,C 0.000} C_DIS
LIN {X -63.840,Y -20.098,Z -214.536,A -90.000,B 90.000,C 0.000} C_DIS
LIN {X -63.207,Y -20.106,Z -214.133,A -90.000,B 90.000,C 0.000} C_DIS
LIN {X -58.096,Y -20.150,Z -210.838,A -90.000,B 90.000,C 0.000} C_DIS
LIN {X -56.163,Y -20.157,Z -209.575,A -90.000,B 90.000,C 0.000} C_DIS
LIN {X -55.798,Y -20.162,Z -209.333,A -90.000,B 90.000,C 0.000} C_DIS
LIN {X -54.974,Y -20.163,Z -208.772,A -90.000,B 90.000,C 0.000} C_DIS
LIN {X -53.223,Y -20.166,Z -207.585,A -90.000,B 90.000,C 0.000} C_DIS
LIN {X -49.786,Y -20.177,Z -205.264,A -90.000,B 90.000,C 0.000} C_DIS
LIN {X -49.386,Y -20.186,Z -204.988,A -90.000,B 90.000,C 0.000} C_DIS
LIN {X -45.599,Y -20.182,Z -202.226,A -90.000,B 90.000,C 0.000} C_DIS
LIN {X -44.481,Y -20.182,Z -201.412,A -90.000,B 90.000,C 0.000} C_DIS
LIN {X -44.324,Y -20.185,Z -201.296,A -90.000,B 90.000,C 0.000} C_DIS
LIN {X -42.534,Y -20.177,Z -199.902,A -90.000,B 90.000,C 0.000} C_DIS
LIN {X -40.078,Y -20.172,Z -197.993,A -90.000,B 90.000,C 0.000} C_DIS
LIN {X -39.894,Y -20.174,Z -197.848,A -90.000,B 90.000,C 0.000} C_DIS
LIN {X -38.300,Y -20.166,Z -196.546,A -90.000,B 90.000,C 0.000} C_DIS
LIN {X -36.380,Y -20.158,Z -194.983,A -90.000,B 90.000,C 0.000} C_DIS
LIN {X -35.835,Y -20.156,Z -194.537,A -90.000,B 90.000,C 0.000} C_DIS
LIN {X -33.054,Y -20.122,Z -192.237,A -90.000,B 90.000,C 0.000} C_DIS
LIN {X -30.708,Y -20.098,Z -190.310,A -90.000,B 90.000,C 0.000} C_DIS
LIN {X -29.859,Y -20.097,Z -189.623,A -90.000,B 90.000,C 0.000} C_DIS
LIN {X -27.984,Y -20.080,Z -188.057,A -90.000,B 90.000,C 0.000} C_DIS
LIN {X -27.104,Y -20.078,Z -187.332,A -90.000,B 90.000,C 0.000} C_DIS
LIN {X -26.997,Y -20.080,Z -187.243,A -90.000,B 90.000,C 0.000} C_DIS
LIN {X -25.164,Y -20.061,Z -185.640,A -90.000,B 90.000,C 0.000} C_DIS
LIN {X -24.573,Y -20.061,Z -185.131,A -90.000,B 90.000,C 0.000} C_DIS
LIN {X -24.408,Y -20.064,Z -184.986,A -90.000,B 90.000,C 0.000} C_DIS
LIN {X -22.817,Y -20.045,Z -183.487,A -90.000,B 90.000,C 0.000} C_DIS
LIN {X -22.043,Y -20.044,Z -182.772,A -90.000,B 90.000,C 0.000} C_DIS
LIN {X -21.947,Y -20.047,Z -182.679,A -90.000,B 90.000,C 0.000} C_DIS
LIN {X -21.092,Y -20.045,Z -181.813,A -90.000,B 90.000,C 0.000} C_DIS
LIN {X -19.524,Y -20.020,Z -180.195,A -90.000,B 90.000,C 0.000} C_DIS
LIN {X -19.444,Y -20.022,Z -180.108,A -90.000,B 90.000,C 0.000} C_DIS
LIN {X -18.771,Y -20.020,Z -179.355,A -90.000,B 90.000,C 0.000} C_DIS
LIN {X -17.370,Y -19.995,Z -177.756,A -90.000,B 90.000,C 0.000} C_DIS
LIN {X -17.234,Y -19.999,Z -177.593,A -90.000,B 90.000,C 0.000} C_DIS
LIN {X -16.773,Y -19.998,Z -177.017,A -90.000,B 90.000,C 0.000} C_DIS
LIN {X -15.210,Y -19.964,Z -175.014,A -90.000,B 90.000,C 0.000} C_DIS
LIN {X -15.031,Y -19.970,Z -174.770,A -90.000,B 90.000,C 0.000} C_DIS
LIN {X -14.678,Y -19.971,Z -174.269,A -90.000,B 90.000,C 0.000} C_DIS
LIN {X -13.428,Y -19.936,Z -172.430,A -90.000,B 90.000,C 0.000} C_DIS
LIN {X -13.250,Y -19.943,Z -172.146,A -90.000,B 90.000,C 0.000} C_DIS
LIN {X -12.850,Y -19.944,Z -171.481,A -90.000,B 90.000,C 0.000} C_DIS
LIN {X -11.806,Y -19.901,Z -169.652,A -90.000,B 90.000,C 0.000} C_DIS
LIN {X -11.659,Y -19.909,Z -169.365,A -90.000,B 90.000,C 0.000} C_DIS
LIN {X -11.498,Y -19.911,Z -169.035,A -90.000,B 90.000,C 0.000} C_DIS
LIN {X -10.598,Y -19.858,Z -167.049,A -90.000,B 90.000,C 0.000} C_DIS
LIN {X -10.469,Y -19.870,Z -166.711,A -90.000,B 90.000,C 0.000} C_DIS
LIN {X -9.894,Y -19.820,Z -164.880,A -90.000,B 90.000,C 0.000} C_DIS
LIN {X -9.841,Y -19.820,Z -164.696,A -90.000,B 90.000,C 0.000} C_DIS
LIN {X -9.784,Y -19.836,Z -164.430,A -90.000,B 90.000,C 0.000} C_DIS
LIN {X -9.584,Y -19.798,Z -162.939,A -90.000,B 90.000,C 0.000} C_DIS
LIN {X -9.585,Y -19.799,Z -162.928,A -90.000,B 90.000,C 0.000} C_DIS
LIN {X -9.710,Y -19.768,Z -162.011,A -90.000,B 90.000,C 0.000} C_DIS
LIN {X -9.754,Y -19.736,Z -161.832,A -90.000,B 90.000,C 0.000} C_DIS
LIN {X -9.844,Y -19.730,Z -161.632,A -90.000,B 90.000,C 0.000} C_DIS
LIN {X -9.910,Y -19.726,Z -161.479,A -90.000,B 90.000,C 0.000} C_DIS
LIN {X -9.960,Y -19.711,Z -161.387,A -90.000,B 90.000,C 0.000} C_DIS
LIN {X -10.156,Y -19.658,Z -161.012,A -90.000,B 90.000,C 0.000} C_DIS
LIN {X -10.388,Y -19.655,Z -160.692,A -90.000,B 90.000,C 0.000} C_DIS
LIN {X -10.601,Y -19.627,Z -160.426,A -90.000,B 90.000,C 0.000} C_DIS
LIN {X -10.758,Y -19.602,Z -160.207,A -90.000,B 90.000,C 0.000} C_DIS
LIN {X -11.272,Y -19.599,Z -159.666,A -90.000,B 90.000,C 0.000} C_DIS
LIN {X -11.385,Y -19.595,Z -159.550,A -90.000,B 90.000,C 0.000} C_DIS
LIN {X -11.802,Y -19.563,Z -159.078,A -90.000,B 90.000,C 0.000} C_DIS
LIN {X -12.300,Y -19.540,Z -158.547,A -90.000,B 90.000,C 0.000} C_DIS
LIN {X -12.463,Y -19.538,Z -158.387,A -90.000,B 90.000,C 0.000} C_DIS
LIN {X -12.666,Y -19.531,Z -158.190,A -90.000,B 90.000,C 0.000} C_DIS
LIN {X -13.024,Y -19.519,Z -157.834,A -90.000,B 90.000,C 0.000} C_DIS
LIN {X -13.622,Y -19.501,Z -157.235,A -90.000,B 90.000,C 0.000} C_DIS
LIN {X -14.104,Y -19.500,Z -156.787,A -90.000,B 90.000,C 0.000} C_DIS
LIN {X -15.374,Y -19.473,Z -155.591,A -90.000,B 90.000,C 0.000} C_DIS
LIN {X -15.960,Y -19.472,Z -155.069,A -90.000,B 90.000,C 0.000} C_DIS
LIN {X -17.692,Y -19.453,Z -153.506,A -90.000,B 90.000,C 0.000} C_DIS
LIN {X -17.762,Y -19.453,Z -153.446,A -90.000,B 90.000,C 0.000} C_DIS
LIN {X -18.262,Y -19.453,Z -153.012,A -90.000,B 90.000,C 0.000} C_DIS
LIN {X -20.557,Y -19.441,Z -151.006,A -90.000,B 90.000,C 0.000} C_DIS
LIN {X -21.130,Y -19.441,Z -150.516,A -90.000,B 90.000,C 0.000} C_DIS
LIN {X -23.417,Y -19.433,Z -148.420,A -90.000,B 90.000,C 0.000} C_DIS
LIN {X -24.277,Y -19.433,Z -147.643,A -90.000,B 90.000,C 0.000} C_DIS
LIN {X -24.426,Y -19.431,Z -147.499,A -90.000,B 90.000,C 0.000} C_DIS
LIN {X -24.631,Y -19.431,Z -147.297,A -90.000,B 90.000,C 0.000} C_DIS
LIN {X -26.504,Y -19.430,Z -145.384,A -90.000,B 90.000,C 0.000} C_DIS
LIN {X -27.909,Y -19.433,Z -143.961,A -90.000,B 90.000,C 0.000} C_DIS
LIN {X -28.055,Y -19.427,Z -143.787,A -90.000,B 90.000,C 0.000} C_DIS
LIN {X -29.374,Y -19.428,Z -142.186,A -90.000,B 90.000,C 0.000} C_DIS
LIN {X -30.940,Y -19.434,Z -140.297,A -90.000,B 90.000,C 0.000} C_DIS
LIN {X -31.243,Y -19.436,Z -139.929,A -90.000,B 90.000,C 0.000} C_DIS
LIN {X -31.409,Y -19.429,Z -139.682,A -90.000,B 90.000,C 0.000} C_DIS
LIN {X -31.507,Y -19.429,Z -139.533,A -90.000,B 90.000,C 0.000} C_DIS
LIN {X -33.588,Y -19.439,Z -136.248,A -90.000,B 90.000,C 0.000} C_DIS
LIN {X -34.003,Y -19.440,Z -135.589,A -90.000,B 90.000,C 0.000} C_DIS
LIN {X -34.173,Y -19.431,Z -135.269,A -90.000,B 90.000,C 0.000} C_DIS
LIN {X -35.172,Y -19.434,Z -133.326,A -90.000,B 90.000,C 0.000} C_DIS
LIN {X -36.246,Y -19.429,Z -131.205,A -90.000,B 90.000,C 0.000} C_DIS
LIN {X -36.394,Y -19.423,Z -130.875,A -90.000,B 90.000,C 0.000} C_DIS
LIN {X -36.771,Y -19.418,Z -130.025,A -90.000,B 90.000,C 0.000} C_DIS
LIN {X -36.934,Y -19.416,Z -129.654,A -90.000,B 90.000,C 0.000} C_DIS
LIN {X -37.537,Y -19.379,Z -128.298,A -90.000,B 90.000,C 0.000} C_DIS
LIN {X -37.885,Y -19.361,Z -127.513,A -90.000,B 90.000,C 0.000} C_DIS
LIN {X -38.125,Y -19.347,Z -126.947,A -90.000,B 90.000,C 0.000} C_DIS
LIN {X -38.505,Y -19.331,Z -126.048,A -90.000,B 90.000,C 0.000} C_DIS
LIN {X -39.063,Y -19.326,Z -124.710,A -90.000,B 90.000,C 0.000} C_DIS
LIN {X -39.166,Y -19.323,Z -124.459,A -90.000,B 90.000,C 0.000} C_DIS
LIN {X -39.275,Y -19.321,Z -124.204,A -90.000,B 90.000,C 0.000} C_DIS
LIN {X -39.778,Y -19.316,Z -123.097,A -90.000,B 90.000,C 0.000} C_DIS
LIN {X -40.227,Y -19.317,Z -122.177,A -90.000,B 90.000,C 0.000} C_DIS
LIN {X -40.497,Y -19.319,Z -121.662,A -90.000,B 90.000,C 0.000} C_DIS
LIN {X -40.649,Y -19.322,Z -121.388,A -90.000,B 90.000,C 0.000} C_DIS
LIN {X -41.104,Y -19.322,Z -120.577,A -90.000,B 90.000,C 0.000} C_DIS
LIN {X -41.470,Y -19.328,Z -120.022,A -90.000,B 90.000,C 0.000} C_DIS
LIN {X -41.582,Y -19.328,Z -119.853,A -90.000,B 90.000,C 0.000} C_DIS
LIN {X -42.082,Y -19.332,Z -119.100,A -90.000,B 90.000,C 0.000} C_DIS
LIN {X -42.557,Y -19.344,Z -118.466,A -90.000,B 90.000,C 0.000} C_DIS
LIN {X -43.017,Y -19.346,Z -117.856,A -90.000,B 90.000,C 0.000} C_DIS
LIN {X -43.266,Y -19.348,Z -117.520,A -90.000,B 90.000,C 0.000} C_DIS
LIN {X -43.848,Y -19.359,Z -116.770,A -90.000,B 90.000,C 0.000} C_DIS
LIN {X -44.387,Y -19.362,Z -116.088,A -90.000,B 90.000,C 0.000} C_DIS
LIN {X -45.727,Y -19.375,Z -114.390,A -90.000,B 90.000,C 0.000} C_DIS
LIN {X -46.233,Y -19.376,Z -113.750,A -90.000,B 90.000,C 0.000} C_DIS
LIN {X -47.034,Y -19.380,Z -112.737,A -90.000,B 90.000,C 0.000} C_DIS
LIN {X -47.520,Y -19.384,Z -112.126,A -90.000,B 90.000,C 0.000} C_DIS
LIN {X -50.083,Y -19.399,Z -108.848,A -90.000,B 90.000,C 0.000} C_DIS
LIN {X -50.431,Y -19.399,Z -108.392,A -90.000,B 90.000,C 0.000} C_DIS
LIN {X -51.319,Y -19.399,Z -107.221,A -90.000,B 90.000,C 0.000} C_DIS
LIN {X -51.917,Y -19.397,Z -106.434,A -90.000,B 90.000,C 0.000} C_DIS
LIN {X -52.683,Y -19.396,Z -105.435,A -90.000,B 90.000,C 0.000} C_DIS
LIN {X -53.062,Y -19.393,Z -104.919,A -90.000,B 90.000,C 0.000} C_DIS
LIN {X -53.583,Y -19.391,Z -104.208,A -90.000,B 90.000,C 0.000} C_DIS
LIN {X -54.618,Y -19.395,Z -102.824,A -90.000,B 90.000,C 0.000} C_DIS
LIN {X -55.162,Y -19.392,Z -102.099,A -90.000,B 90.000,C 0.000} C_DIS
LIN {X -55.715,Y -19.387,Z -101.347,A -90.000,B 90.000,C 0.000} C_DIS
LIN {X -55.963,Y -19.387,Z -101.007,A -90.000,B 90.000,C 0.000} C_DIS
LIN {X -56.578,Y -19.384,Z -100.167,A -90.000,B 90.000,C 0.000} C_DIS
LIN {X -57.126,Y -19.383,Z -99.442,A -90.000,B 90.000,C 0.000} C_DIS
LIN {X -57.921,Y -19.386,Z -98.386,A -90.000,B 90.000,C 0.000} C_DIS
LIN {X -59.356,Y -19.387,Z -96.476,A -90.000,B 90.000,C 0.000} C_DIS
LIN {X -59.817,Y -19.384,Z -95.861,A -90.000,B 90.000,C 0.000} C_DIS
LIN {X -60.689,Y -19.384,Z -94.722,A -90.000,B 90.000,C 0.000} C_DIS
LIN {X -62.099,Y -19.384,Z -92.924,A -90.000,B 90.000,C 0.000} C_DIS
LIN {X -62.360,Y -19.388,Z -92.602,A -90.000,B 90.000,C 0.000} C_DIS
LIN {X -63.951,Y -19.387,Z -90.629,A -90.000,B 90.000,C 0.000} C_DIS
LIN {X -64.207,Y -19.390,Z -90.326,A -90.000,B 90.000,C 0.000} C_DIS
LIN {X -65.244,Y -19.386,Z -89.104,A -90.000,B 90.000,C 0.000} C_DIS
LIN {X -65.596,Y -19.387,Z -88.694,A -90.000,B 90.000,C 0.000} C_DIS
LIN {X -65.936,Y -19.391,Z -88.315,A -90.000,B 90.000,C 0.000} C_DIS
LIN {X -67.349,Y -19.390,Z -86.752,A -90.000,B 90.000,C 0.000} C_DIS
LIN {X -67.433,Y -19.391,Z -86.664,A -90.000,B 90.000,C 0.000} C_DIS
LIN {X -68.124,Y -19.397,Z -85.945,A -90.000,B 90.000,C 0.000} C_DIS
LIN {X -69.095,Y -19.398,Z -84.912,A -90.000,B 90.000,C 0.000} C_DIS
LIN {X -70.543,Y -19.409,Z -83.424,A -90.000,B 90.000,C 0.000} C_DIS
LIN {X -70.918,Y -19.411,Z -83.036,A -90.000,B 90.000,C 0.000} C_DIS
LIN {X -71.118,Y -19.414,Z -82.836,A -90.000,B 90.000,C 0.000} C_DIS
LIN {X -72.400,Y -19.426,Z -81.574,A -90.000,B 90.000,C 0.000} C_DIS
LIN {X -72.874,Y -19.439,Z -81.144,A -90.000,B 90.000,C 0.000} C_DIS
LIN {X -73.241,Y -19.445,Z -80.813,A -90.000,B 90.000,C 0.000} C_DIS
LIN {X -73.926,Y -19.455,Z -80.198,A -90.000,B 90.000,C 0.000} C_DIS
LIN {X -73.977,Y -19.456,Z -80.155,A -90.000,B 90.000,C 0.000} C_DIS
LIN {X -74.354,Y -19.476,Z -79.866,A -90.000,B 90.000,C 0.000} C_DIS
LIN {X -74.899,Y -19.494,Z -79.456,A -90.000,B 90.000,C 0.000} C_DIS
LIN {X -75.320,Y -19.540,Z -79.237,A -90.000,B 90.000,C 0.000} C_DIS
LIN {X -75.545,Y -19.544,Z -79.131,A -90.000,B 90.000,C 0.000} C_DIS
LIN {X -75.827,Y -19.527,Z -79.013,A -90.000,B 90.000,C 0.000} C_DIS
LIN {X -75.917,Y -19.520,Z -78.976,A -90.000,B 90.000,C 0.000} C_DIS
LIN {X -75.954,Y -19.519,Z -78.966,A -90.000,B 90.000,C 0.000} C_DIS
LIN {X -76.854,Y -19.468,Z -78.725,A -90.000,B 90.000,C 0.000} C_DIS
LIN {X -77.020,Y -19.462,Z -78.689,A -90.000,B 90.000,C 0.000} C_DIS
LIN {X -77.474,Y -19.446,Z -78.572,A -90.000,B 90.000,C 0.000} C_DIS
LIN {X -78.071,Y -19.441,Z -78.412,A -90.000,B 90.000,C 0.000} C_DIS
LIN {X -78.548,Y -19.433,Z -78.267,A -90.000,B 90.000,C 0.000} C_DIS
LIN {X -78.654,Y -19.430,Z -78.230,A -90.000,B 90.000,C 0.000} C_DIS
LIN {X -79.197,Y -19.417,Z -78.035,A -90.000,B 90.000,C 0.000} C_DIS
LIN {X -79.776,Y -19.419,Z -77.818,A -90.000,B 90.000,C 0.000} C_DIS
LIN {X -80.444,Y -19.424,Z -77.568,A -90.000,B 90.000,C 0.000} C_DIS
LIN {X -80.664,Y -19.429,Z -77.485,A -90.000,B 90.000,C 0.000} C_DIS
LIN {X -80.713,Y -19.428,Z -77.462,A -90.000,B 90.000,C 0.000} C_DIS
LIN {X -81.188,Y -19.427,Z -77.226,A -90.000,B 90.000,C 0.000} C_DIS
LIN {X -81.673,Y -19.425,Z -76.961,A -90.000,B 90.000,C 0.000} C_DIS
LIN {X -82.657,Y -19.435,Z -76.417,A -90.000,B 90.000,C 0.000} C_DIS
LIN {X -82.985,Y -19.433,Z -76.211,A -90.000,B 90.000,C 0.000} C_DIS
LIN {X -83.350,Y -19.435,Z -75.974,A -90.000,B 90.000,C 0.000} C_DIS
LIN {X -83.589,Y -19.439,Z -75.816,A -90.000,B 90.000,C 0.000} C_DIS
LIN {X -84.596,Y -19.452,Z -75.112,A -90.000,B 90.000,C 0.000} C_DIS
LIN {X -84.824,Y -19.455,Z -74.944,A -90.000,B 90.000,C 0.000} C_DIS
LIN {X -85.183,Y -19.464,Z -74.672,A -90.000,B 90.000,C 0.000} C_DIS
LIN {X -85.621,Y -19.475,Z -74.331,A -90.000,B 90.000,C 0.000} C_DIS
LIN {X -85.847,Y -19.485,Z -74.165,A -90.000,B 90.000,C 0.000} C_DIS
LIN {X -86.074,Y -19.492,Z -73.994,A -90.000,B 90.000,C 0.000} C_DIS
LIN {X -86.480,Y -19.498,Z -73.703,A -90.000,B 90.000,C 0.000} C_DIS
LIN {X -86.812,Y -19.511,Z -73.460,A -90.000,B 90.000,C 0.000} C_DIS
LIN {X -87.112,Y -19.519,Z -73.232,A -90.000,B 90.000,C 0.000} C_DIS
LIN {X -87.452,Y -19.522,Z -72.964,A -90.000,B 90.000,C 0.000} C_DIS
LIN {X -87.557,Y -19.525,Z -72.888,A -90.000,B 90.000,C 0.000} C_DIS
LIN {X -88.044,Y -19.522,Z -72.491,A -90.000,B 90.000,C 0.000} C_DIS
LIN {X -88.272,Y -19.525,Z -72.313,A -90.000,B 90.000,C 0.000} C_DIS
LIN {X -88.700,Y -19.525,Z -71.964,A -90.000,B 90.000,C 0.000} C_DIS
LIN {X -89.053,Y -19.519,Z -71.651,A -90.000,B 90.000,C 0.000} C_DIS
LIN {X -89.354,Y -19.523,Z -71.377,A -90.000,B 90.000,C 0.000} C_DIS
LIN {X -89.646,Y -19.522,Z -71.096,A -90.000,B 90.000,C 0.000} C_DIS
LIN {X -90.003,Y -19.527,Z -70.747,A -90.000,B 90.000,C 0.000} C_DIS
LIN {X -90.188,Y -19.532,Z -70.572,A -90.000,B 90.000,C 0.000} C_DIS
LIN {X -90.668,Y -19.537,Z -70.099,A -90.000,B 90.000,C 0.000} C_DIS
LIN {X -90.829,Y -19.544,Z -69.954,A -90.000,B 90.000,C 0.000} C_DIS
LIN {X -91.251,Y -19.546,Z -69.559,A -90.000,B 90.000,C 0.000} C_DIS
LIN {X -91.520,Y -19.556,Z -69.330,A -90.000,B 90.000,C 0.000} C_DIS
LIN {X -91.717,Y -19.558,Z -69.165,A -90.000,B 90.000,C 0.000} C_DIS
LIN {X -92.034,Y -19.570,Z -68.927,A -90.000,B 90.000,C 0.000} C_DIS
LIN {X -92.371,Y -19.579,Z -68.678,A -90.000,B 90.000,C 0.000} C_DIS
LIN {X -92.537,Y -19.580,Z -68.547,A -90.000,B 90.000,C 0.000} C_DIS
LIN {X -93.267,Y -19.599,Z -68.016,A -90.000,B 90.000,C 0.000} C_DIS
LIN {X -93.352,Y -19.600,Z -67.951,A -90.000,B 90.000,C 0.000} C_DIS
LIN {X -93.491,Y -19.606,Z -67.854,A -90.000,B 90.000,C 0.000} C_DIS
LIN {X -93.821,Y -19.611,Z -67.609,A -90.000,B 90.000,C 0.000} C_DIS
LIN {X -94.410,Y -19.626,Z -67.166,A -90.000,B 90.000,C 0.000} C_DIS
LIN {X -94.832,Y -19.627,Z -66.828,A -90.000,B 90.000,C 0.000} C_DIS
LIN {X -95.315,Y -19.638,Z -66.439,A -90.000,B 90.000,C 0.000} C_DIS
LIN {X -95.506,Y -19.640,Z -66.280,A -90.000,B 90.000,C 0.000} C_DIS
LIN {X -95.983,Y -19.644,Z -65.879,A -90.000,B 90.000,C 0.000} C_DIS
LIN {X -96.545,Y -19.655,Z -65.408,A -90.000,B 90.000,C 0.000} C_DIS
LIN {X -97.033,Y -19.657,Z -64.991,A -90.000,B 90.000,C 0.000} C_DIS
LIN {X -97.551,Y -19.664,Z -64.562,A -90.000,B 90.000,C 0.000} C_DIS
LIN {X -97.986,Y -19.661,Z -64.206,A -90.000,B 90.000,C 0.000} C_DIS
LIN {X -98.250,Y -19.663,Z -63.996,A -90.000,B 90.000,C 0.000} C_DIS
LIN {X -98.962,Y -19.645,Z -63.449,A -90.000,B 90.000,C 0.000} C_DIS
LIN {X -99.222,Y -19.643,Z -63.255,A -90.000,B 90.000,C 0.000} C_DIS
LIN {X -99.892,Y -19.627,Z -62.761,A -90.000,B 90.000,C 0.000} C_DIS
LIN {X -100.268,Y -19.625,Z -62.482,A -90.000,B 90.000,C 0.000} C_DIS
LIN {X -100.853,Y -19.626,Z -62.043,A -90.000,B 90.000,C 0.000} C_DIS
LIN {X -101.288,Y -19.632,Z -61.726,A -90.000,B 90.000,C 0.000} C_DIS
LIN {X -102.295,Y -19.657,Z -60.941,A -90.000,B 90.000,C 0.000} C_DIS
